			(* Spindel mit Ausfahrgeschwindigkeit *)
			IF ptrTAxisS^.T_CtrleSingle.xNotMoving THEN
				ptrTAxisS^.T_CtrleSingle.iFunction:=6;	(* Move Velocity *)
			ELSE
				ptrTAxisS^.T_CtrleSingle.iFunction:=12;	(* Move Velocity *)
			END_IF;
			ptrTAxisS^.T_CtrleSingle.lrVelocity:=T_Station_Parameter.T_StProcess.rOutfeedSpindleSpeed;
			ptrTAxisS^.T_CtrleSingle.xExecute:=TRUE;
			IF NOT(ptrTAxisBubbler^.T_CtrleDCAxis.xNotMoving) THEN
				(* Abstreifer ZU *)
				QxCylStripperClose_St1:=TRUE;
				QxCylStripperOpen_St1:=FALSE;
			END_IF
		END_IF;
		IF ptrTAxisZ^.T_LiveValue.lrActualPosition <= grZ_LoadPos THEN
			rStFct_CtrlInputWorkingSpeed:=0.0;
			T_Z_St1_Ctrle.diVelocityCommandValue:=0; (* Make sure Z axis is not moving anymore *)

			 IF ptrTAxisS^.T_CtrleSingle.xExecute AND ptrTAxisS^.T_CtrleSingle.xDone THEN
				xStFct_StartMainPrc:=FALSE;
				xStFct_InitStep:=FALSE;
				iStFct_StepPrc:=iStFct_StepPrc + 1;
			END_IF;
		END_IF;

	61: 	(* Prozess end, reset Z axis *)
		IF NOT(xStFct_InitStep) THEN
			xStFct_InitStep:=TRUE;
			xStFct_OutfeedStrokeRunning:=FALSE;
			ptrTAxisZ^.T_CtrleSingle.iFunction:=1;
			ptrTAxisZ^.T_CtrleSingle.xExecute:=TRUE;
			IF NOT(ptrTAxisBubbler^.T_CtrleDCAxis.xNotMoving) THEN
				(* Abstreifer ZU *)
				QxCylStripperClose_St1:=TRUE;
				QxCylStripperOpen_St1:=FALSE;
			END_IF
		END_IF;
		IF NOT(ptrTAxisZ^.T_CtrleSingle.xExecute) AND ptrTAxisZ^.T_CtrleSingle.xDone THEN
			xStFct_StartMainPrc:=FALSE;
			xStFct_InitStep:=FALSE;
			iStFct_StepPrc:=0;
			xStFct_SetEnd:=TRUE;
			IF xProcessDone THEN
				IF (NOT(ptrTAxisS^.T_CtrleSingle.xNotMoving) OR NOT(ptrTAxisS^.T_CtrleSingle.xDone)) AND
				     NOT((ptrTAxisS^.T_CtrleSingle.iFunction = 5) AND NOT(ptrTAxisS^.T_CtrleSingle.xDone)) AND NOT(ptrTAxisS^.T_CtrleSingle.xErr) THEN
					ptrTAxisS^.T_CtrleSingle.iFunction:=5;
					ptrTAxisS^.T_CtrleSingle.xExecute:=TRUE;
				END_IF;
			END_IF;
			(* Abstreifer AUF *)
			QxCylStripperClose_St1:=FALSE;
			QxCylStripperOpen_St1:=TRUE;
		END_IF;

		(* Dies gilt für den neuen Ablauf und setzt die Z Achse zurück auf die LadePos und gibt einen Fehler aus *)
	90:	IF (T_Station_Parameter.T_StProcess.rZ1AxisPosSwitchOAxisOff >= garPositionEndProcCalc[1])
		OR ((ptrTAxisZ^.T_LiveValue.lrActualPosition <= T_Station_Parameter.T_StProcess.rZ1AxisPosSwitchOAxisOff)
		OR (ABS(ptrTAxisZ^.T_LiveValue.lrActualPosition - T_Station_Parameter.T_StProcess.rPositionLoad) <= 10.0)) THEN
			QxFastStrokeOn_St1:=FALSE;
		END_IF;
		IF NOT(xStFct_InitStep) THEN
			xStFct_InitStep:=TRUE;
			ptrTAxisZ^.T_CtrleSingle.iFunction:=7;	(* Absolut Bewegung *)
			ptrTAxisZ^.T_CtrleSingle.lrPosition:=grZ_LoadPos;	(* AxisSlide auf BearbStartPosition setzen *)
			ptrTAxisZ^.T_CtrleSingle.lrVelocity:=rOutfeedStrokeAxisSpeed;
			ptrTAxisZ^.T_CtrleSingle.xExecute:=TRUE;
			(* Spindel mit Ausfahrgeschwindigkeit *)
			IF ptrTAxisS^.T_CtrleSingle.xNotMoving THEN
				ptrTAxisS^.T_CtrleSingle.iFunction:=6;	(* Move Velocity *)
			ELSE
				ptrTAxisS^.T_CtrleSingle.iFunction:=12;	(* Move Velocity *)
			END_IF;
			ptrTAxisS^.T_CtrleSingle.lrVelocity:=T_Station_Parameter.T_StProcess.rOutfeedSpindleSpeed;
			ptrTAxisS^.T_CtrleSingle.xExecute:=TRUE;
			IF NOT(ptrTAxisBubbler^.T_CtrleDCAxis.xNotMoving) THEN
				(* Abstreifer ZU *)
				QxCylStripperClose_St1:=TRUE;
				QxCylStripperOpen_St1:=FALSE;
			END_IF
		END_IF;
		IF NOT(ptrTAxisZ^.T_CtrleSingle.xExecute) AND ptrTAxisZ^.T_CtrleSingle.xDone AND
		     NOT(ptrTAxisS^.T_CtrleSingle.xExecute) AND ptrTAxisS^.T_CtrleSingle.xDone THEN
			xStFct_StartMainPrc:=FALSE;
			xStFct_InitStep:=FALSE;
			iStFct_StepPrc:=iStFct_StepPrc + 1;
		END_IF;

	91:	(* Abstreifer AUF *)
		QxCylStripperClose_St1:=FALSE;
		QxCylStripperOpen_St1:=TRUE;
		QxFastStrokeOn_St1:=FALSE;
		xStFct_HardwareError:=TRUE;
		diStFct_TmpErrorNr:=44;		(* Beim zylindrischer Teil wurde die Max EndPos erreicht *)

	END_CASE;
END_IF;
(******************************************************************************************************************************************)
(****************************			             Stationsfunktion Parallelablauf                                       *****************************)
(******************************************************************************************************************************************)

(******************************************************************************************************************************************)
(****************************				     Stationsfunktion Endprozedur                                    *****************************)
(******************************************************************************************************************************************)
StationFunction_Ctrl_End;
END_ACTION
ACTION StationFunction_Fct_06_ToolRotationOFF:
(******************************************************************************************************************************************)
(****************************				           Reset Stationsfunktion                                            *****************************)
(******************************************************************************************************************************************)
StationFunction_Ctrl_Reset;
(******************************************************************************************************************************************)
(****************************			        Stationsfunktion Fehler Controller                                    *****************************)
(******************************************************************************************************************************************)
StationFunction_Ctrl_Error;
(******************************************************************************************************************************************)
(****************************				    Stationsfunktion Haupt Controller                               *****************************)
(******************************************************************************************************************************************)
StationFunction_Ctrl_Main;
(******************************************************************************************************************************************)
(****************************			         Stationsfunktion sofort Unterbrechung                           *****************************)
(******************************************************************************************************************************************)
StationFunction_Ctrl_Stop;
(******************************************************************************************************************************************)
(****************************			             Stationsfunktion Hauptablauf                                       *****************************)
(******************************************************************************************************************************************)
IF xStFct_StartMainPrc AND NOT(xStFct_SetEnd) AND NOT(xStFct_HardwareError) AND NOT(xStFct_TmpStop) THEN
	CASE iStFct_StepPrc OF
	1:	IF NOT(xStFct_InitStep) THEN
			IF NOT(ptrTAxisS^.T_CtrleSingle.xNotMoving) AND ptrTAxisS^.T_CtrleSingle.xPower THEN
				(* Die Spindel dreht, daher muss sie gestoppt werden und dann der Strom noch ausschalten *)
				iStFct_StepPrc:=iStFct_StepPrc + 1;
			ELSIF ptrTAxisS^.T_CtrleSingle.xNotMoving AND ptrTAxisS^.T_CtrleSingle.xPower THEN
				(* Die Spindel ist schon gestoppt, der Strom muss aber noch ausgeschaltet werden *)
				iStFct_StepPrc:=3;
			ELSE
				(* Die Spindel ist schon im entsprechenden Zustand, daher kann die Funktion beendet werden *)
				iStFct_StepPrc:=4;
			END_IF;
			xStFct_StartMainPrc:=FALSE;
			xStFct_InitStep:=FALSE;
		END_IF;
	2:	IF NOT(xStFct_InitStep) THEN
			xStFct_InitStep:=TRUE;
			ptrTAxisS^.T_CtrleSingle.iFunction:=5;
			ptrTAxisS^.T_CtrleSingle.xExecute:=TRUE;
		END_IF;
		IF NOT(ptrTAxisS^.T_CtrleSingle.xExecute) AND ptrTAxisS^.T_CtrleSingle.xDone AND ptrTAxisS^.T_CtrleSingle.xNotMoving THEN
			xStFct_StartMainPrc:=FALSE;
			xStFct_InitStep:=FALSE;
			iStFct_StepPrc:=iStFct_StepPrc + 1;
		END_IF;
	3:	IF NOT(xStFct_InitStep) THEN
			xStFct_InitStep:=TRUE;
			ptrTAxisS^.T_CtrleSingle.iFunction:=4;	(* Strom ausschalten *)
			ptrTAxisS^.T_CtrleSingle.xExecute:=TRUE;
		END_IF;
		IF NOT(ptrTAxisS^.T_CtrleSingle.xExecute) AND ptrTAxisS^.T_CtrleSingle.xDone AND NOT(ptrTAxisS^.T_CtrleSingle.xPower) THEN
			xStFct_StartMainPrc:=FALSE;
			xStFct_InitStep:=FALSE;
			iStFct_StepPrc:=iStFct_StepPrc + 1;
		END_IF;
	4:	xStFct_StartMainPrc:=FALSE;
		xStFct_InitStep:=FALSE;
		iStFct_StepPrc:=0;
		xStFct_SetEnd:=TRUE;
	END_CASE;
END_IF;
(******************************************************************************************************************************************)
(****************************			             Stationsfunktion Parallelablauf                                       *****************************)
(******************************************************************************************************************************************)
IF xStFct_StartPrc_Parallel AND NOT(xStFct_SetEnd) AND NOT(xStFct_HardwareError) THEN
	CASE iStFct_StepPrc_Parallel OF
	1:	iStFct_StepPrc_Parallel:=1;
		xStFct_InitStep_Parallel:=FALSE;
		xStFct_StartPrc_Parallel:=FALSE;
	END_CASE;
END_IF;
(******************************************************************************************************************************************)
(****************************				     Stationsfunktion Endprozedur                                    *****************************)
(******************************************************************************************************************************************)
StationFunction_Ctrl_End;
END_ACTION
ACTION StationFunction_Fct_07_Calibration:
(******************************************************************************************************************************************)
(****************************				           Reset Stationsfunktion                                            *****************************)
(******************************************************************************************************************************************)
StationFunction_Ctrl_Reset;
(******************************************************************************************************************************************)
(****************************			        Stationsfunktion Fehler Controller                                    *****************************)
(******************************************************************************************************************************************)
StationFunction_Ctrl_Error;
(******************************************************************************************************************************************)
(****************************				    Stationsfunktion Haupt Controller                               *****************************)
(******************************************************************************************************************************************)
StationFunction_Ctrl_Main;
(******************************************************************************************************************************************)
(****************************			         Stationsfunktion sofort Unterbrechung                           *****************************)
(******************************************************************************************************************************************)
StationFunction_Ctrl_Stop;
(******************************************************************************************************************************************)
(****************************			             Stationsfunktion Hauptablauf                                       *****************************)
(******************************************************************************************************************************************)
IF xStFct_TmpStop AND NOT(xStFct_HardwareError) THEN
	T_Station_Parameter.T_Fct_SpindleCalibration.arOffsetToolDeflection[1]:=rStFct_TmpOffsetDeflection;
	T_Station_Parameter.T_Fct_SpindleCalibration.arOffsetToolTorque[1]:=rStFct_TmpOffsetTorque;
END_IF;
IF xStFct_StartMainPrc AND NOT(xStFct_SetEnd) AND NOT(xStFct_HardwareError) AND NOT(xStFct_TmpStop) THEN
	IF ((iStFct_StepPrc >= 4) AND (iStFct_StepPrc <= 6)) OR xStFct_StartPrc_Parallel THEN
		IF ((iStFct_StepPrc >= 4) AND (iStFct_StepPrc <= 6)) THEN
			T_Station_Work.THWWorkStation.TCtrlWork.rOffsetToolDeflection:=rStFct_ForceDeflection;
		END_IF;
		IF xStFct_StartPrc_Parallel THEN
			T_Station_Work.THWWorkStation.TCtrlWork.rOffsetToolTorque:=rStFct_ForceTorque;
		END_IF;
		CASE T_ExchgParam.bToolSpindleActive OF
		1:	(* Maxon Spindel *)
			IF NOT(xStFct_DeflCalibError) AND ((rStFct_ForceDeflection < 0) OR (rStFct_ForceDeflection > (T_Station_Parameter.T_SpindleSystem.rMaxDeflectionForce + rStFct_TmpOffsetDeflection))) THEN
				xStFct_DeflCalibError:=TRUE;
				xStFct_StartMainPrc:=FALSE;
				xStFct_InitStep:=FALSE;
				iStFct_StepPrc:=7;
				T_Station_Parameter.T_Fct_SpindleCalibration.arOffsetToolDeflection[1]:=rStFct_TmpOffsetDeflection;
			END_IF;
			IF NOT(xStFct_TorqueCalibError) AND ((rStFct_ForceTorque < 0) OR (rStFct_ForceTorque > (T_Station_Parameter.T_TorqueSystem.rMaxTorque_HC + rStFct_TmpOffsetTorque))) THEN
				xStFct_TorqueCalibError:=TRUE;
				xStFct_StartMainPrc:=FALSE;
				xStFct_InitStep:=FALSE;
				iStFct_StepPrc:=7;
				T_Station_Parameter.T_Fct_SpindleCalibration.arOffsetToolTorque[1]:=rStFct_TmpOffsetTorque;
				xStFct_StartPrc_Parallel:=FALSE;
			END_IF;
		2:	(* Beckhoff Spindel L *)
			IF NOT(xStFct_DeflCalibError) AND ((rStFct_ForceDeflection < 0) OR (rStFct_ForceDeflection > (T_Station_Parameter.T_SpindleSystem_L.rMaxDeflectionForce + rStFct_TmpOffsetDeflection))) THEN
				xStFct_DeflCalibError:=TRUE;
				xStFct_StartMainPrc:=FALSE;
				xStFct_InitStep:=FALSE;
				iStFct_StepPrc:=7;
				T_Station_Parameter.T_Fct_SpindleCalibration.arOffsetToolDeflection[1]:=rStFct_TmpOffsetDeflection;
			END_IF;
		3:	(* Beckhoff Spindel M *)
			IF NOT(xStFct_DeflCalibError) AND ((rStFct_ForceDeflection < 0) OR (rStFct_ForceDeflection > (T_Station_Parameter.T_SpindleSystem_M.rMaxDeflectionForce + rStFct_TmpOffsetDeflection))) THEN
				xStFct_DeflCalibError:=TRUE;
				xStFct_StartMainPrc:=FALSE;
				xStFct_InitStep:=FALSE;
				iStFct_StepPrc:=7;
				T_Station_Parameter.T_Fct_SpindleCalibration.arOffsetToolDeflection[1]:=rStFct_TmpOffsetDeflection;
			END_IF;
		END_CASE;
	END_IF;
	IF T_Station_Work.THWWorkStation.TCtrlWork.xWorkStopToolRotation THEN
		xStFct_TmpSaveOffset:=FALSE;
		xStFct_StartMainPrc:=FALSE;
		xStFct_InitStep:=FALSE;
		iStFct_StepPrc:=0;
		xStFct_SetEnd:=TRUE;
	END_IF;
	(* Deflection Sensor ON/OFF-->Muss für 0.1s gesetzt bleiben, damit Sensor ON/OFF ist, damit Prellungen ausgeschaltet werden können *)
	IF ptrTCylToolDeflection^.T_CtrleCyl.xStatePosOn THEN
		TONStFct_DeflectionSensorOFF(IN:=FALSE);
		TONStFct_DeflectionSensorON(IN:=TRUE,PT:=T#0.05s);
		IF TONStFct_DeflectionSensorON.Q THEN
			xStFct_DeflectionSensorON:=TRUE;
		END_IF;
	ELSE
		TONStFct_DeflectionSensorON(IN:=FALSE);
		TONStFct_DeflectionSensorOFF(IN:=TRUE,PT:=T#0.05s);
		IF TONStFct_DeflectionSensorOFF.Q THEN
			xStFct_DeflectionSensorON:=FALSE;
		END_IF;
	END_IF;
	(* Toruque Sensor ON/OFF-->Muss für 0.1s gesetzt bleiben, damit Sensor ON/OFF ist, damit Prellungen ausgeschaltet werden können *)
	IF ptrTCylToolTorqueHC^.T_CtrleCyl.xStatePosOn THEN
		TONStFct_TorqueSensorOFF(IN:=FALSE);
		TONStFct_TorqueSensorON(IN:=TRUE,PT:=T#0.04s);
		IF TONStFct_TorqueSensorON.Q THEN
			xStFct_TorqueSensorON:=TRUE;
		END_IF;
	ELSE
		TONStFct_TorqueSensorON(IN:=FALSE);
		TONStFct_TorqueSensorOFF(IN:=TRUE,PT:=T#0.04s);
		IF TONStFct_TorqueSensorOFF.Q THEN
			xStFct_TorqueSensorON:=FALSE;
		END_IF;
	END_IF;
	CASE iStFct_StepPrc OF
	1:	(* Offsets während Kalibrierung auf 0 setzen, aktuelle Werte für den Fehlerfall temporär ziwschen speichern*)
		xStFct_TmpSaveOffset:=TRUE;
		TONStFct_DeflectionSensorON(IN:=FALSE);
		TONStFct_DeflectionSensorOFF(IN:=FALSE);
		TONStFct_TorqueSensorON(IN:=FALSE);
		TONStFct_TorqueSensorOFF(IN:=FALSE);
		xStFct_DeflectionSensorON:=FALSE;
		xStFct_TorqueSensorON:=FALSE;
		IF  (T_Station_Parameter.T_Fct_SpindleCalibration.arOffsetToolDeflection[1] < 0) THEN
			T_Station_Parameter.T_Fct_SpindleCalibration.arOffsetToolDeflection[1]:=2.0;
			rStFct_TmpOffsetDeflection:= 2.0;
		ELSE
			rStFct_TmpOffsetDeflection:= T_Station_Parameter.T_Fct_SpindleCalibration.arOffsetToolDeflection[1];
		END_IF;
		IF (T_Station_Parameter.T_Fct_SpindleCalibration.arOffsetToolTorque[1] < 0) THEN
			T_Station_Parameter.T_Fct_SpindleCalibration.arOffsetToolTorque[1]:=2.0;
			rStFct_TmpOffsetTorque:= 2.0;
		ELSE
			rStFct_TmpOffsetTorque:= T_Station_Parameter.T_Fct_SpindleCalibration.arOffsetToolTorque[1];
		END_IF;
		xStFct_DeflCalibError:=FALSE;
		xStFct_TorqueCalibError:=FALSE;
		IF NOT(xStFct_InitStep) THEN
			(* Falls die Spindel nicht bestromt ist, dann wird der Motorstrom eingeschaltet *)
			IF NOT(ptrTAxisS^.T_CtrleSingle.xPower) THEN
				ptrTAxisS^.T_CtrleSingle.iFunction:=3;	(* Strom einschalten *)
				ptrTAxisS^.T_CtrleSingle.xExecute:=TRUE;
			END_IF;
			(* Zylinder für Überlast Drehmoment *)
			ptrTCylToolTorqueOverload^.T_CtrleCyl.iFunction:=2;
			ptrTCylToolTorqueOverload^.T_Config.tDelayOn:=T#0.2s;
			CASE T_ExchgParam.bToolSpindleActive OF
			1:	(* Maxon Spindel *)
				ptrTCylToolTorqueOverload^.T_CtrleCyl.T_Analog.rForceIn:=T_Station_Parameter.T_TorqueSystem.rMaxTorque_HCOver;	(* Dieser Zylinder muss aktiviert sein, anderenfalls führt es zu Probleme mit der Kalibrierung wegem auskoppeln der Spindel *)
			END_CASE;
			ptrTCylToolTorqueOverload^.T_CtrleCyl.xExecute:=(T_ExchgParam.bToolSpindleActive = 1);		(* nur ausführen wenn Maxon Spindel aktiv ist *)
			xStFct_InitStep:=TRUE;
		END_IF;
		IF NOT(ptrTAxisS^.T_CtrleSingle.xExecute) AND ptrTAxisS^.T_CtrleSingle.xDone AND ptrTAxisS^.T_CtrleSingle.xPower AND
		     NOT(ptrTCylToolTorqueOverload^.T_CtrleCyl.xExecute) AND ptrTCylToolTorqueOverload^.T_CtrleCyl.xDone THEN
			IF T_Station_Work.THWWorkStation.TCtrlWork.xActiveCalibrateToolDeflection THEN
				FOR iStFct_ii:=5 TO 2 BY -1 DO
					T_Station_Parameter.T_Fct_SpindleCalibration.arOffsetToolDeflection[iStFct_ii]:=T_Station_Parameter.T_Fct_SpindleCalibration.arOffsetToolDeflection[iStFct_ii-1];
				END_FOR;
			END_IF;
			IF T_Station_Work.THWWorkStation.TCtrlWork.xActiveCalibrateToolTorque THEN
				FOR iStFct_ii:=5 TO 2 BY -1 DO
					T_Station_Parameter.T_Fct_SpindleCalibration.arOffsetToolTorque[iStFct_ii]:=T_Station_Parameter.T_Fct_SpindleCalibration.arOffsetToolTorque[iStFct_ii-1];
				END_FOR;
			END_IF;
			xStFct_StartMainPrc:=FALSE;
			xStFct_InitStep:=FALSE;
			iStFct_StepPrc:=iStFct_StepPrc + 1;
		END_IF;
	2:	IF NOT(xStFct_InitStep) THEN
			xStFct_InitStep:=TRUE;
			IF ptrTAxisS^.T_CtrleSingle.xNotMoving THEN
				ptrTAxisS^.T_CtrleSingle.iFunction:=6;	(* Move Velocity *)
			ELSE
				ptrTAxisS^.T_CtrleSingle.iFunction:=12;	(* Move Velocity with new velocity *)
			END_IF;
			ptrTAxisS^.T_CtrleSingle.lrVelocity:=T_Station_Parameter.T_OnlineChange.rWorkingSpindleSpeed;
			ptrTAxisS^.T_CtrleSingle.xExecute:=TRUE;
		END_IF;
		IF NOT(ptrTAxisS^.T_CtrleSingle.xExecute) AND ptrTAxisS^.T_CtrleSingle.xDone AND NOT(ptrTAxisS^.T_CtrleSingle.xNotMoving) THEN
			rStFct_ForceDeflection:=rStFct_TmpOffsetDeflection;
			rStFct_ForceTorque:=rStFct_TmpOffsetTorque;
			IF T_Station_Work.THWWorkStation.TCtrlWork.xActiveCalibrateToolDeflection THEN
				T_Station_Parameter.T_Fct_SpindleCalibration.arOffsetToolDeflection[1]:=0.0;
			END_IF;
			IF T_Station_Work.THWWorkStation.TCtrlWork.xActiveCalibrateToolTorque THEN
				T_Station_Parameter.T_Fct_SpindleCalibration.arOffsetToolTorque[1]:=0.0;
			END_IF;
			xStFct_StartMainPrc:=FALSE;
			xStFct_InitStep:=FALSE;
			iStFct_StepPrc:=iStFct_StepPrc + 1;
		END_IF;
	(* Überprüfe zuerst ob die Sensorik in Ordnung ist *)
	3:	IF NOT(xStFct_InitStep) THEN
			xStFct_InitStep:=TRUE;
			IF T_Station_Work.THWWorkStation.TCtrlWork.xActiveCalibrateToolDeflection THEN
				(* Zylinder für Auslenkung-->ausschalten *)
				ptrTCylToolDeflection^.T_CtrleCyl.iFunction:=1;
				ptrTCylToolDeflection^.T_CtrleCyl.T_Analog.tDelayActiv:=T#0s;
				ptrTCylToolDeflection^.T_Config.tDelayOff:=T#0.3s;
				ptrTCylToolDeflection^.T_Config.xCtrlePosOff:=FALSE;
				ptrTCylToolDeflection^.T_CtrleCyl.T_Analog.rForceIn:=0.0;
				ptrTCylToolDeflection^.T_CtrleCyl.xExecute:=TRUE;
			END_IF;
			IF T_Station_Work.THWWorkStation.TCtrlWork.xActiveCalibrateToolTorque THEN
				(* Zylinder für Drehmoment-->ausschalten *)
				ptrTCylToolTorqueHC^.T_CtrleCyl.iFunction:=1;
				ptrTCylToolTorqueHC^.T_CtrleCyl.T_Analog.tDelayActiv:=T#0s;
				ptrTCylToolTorqueHC^.T_Config.tDelayOff:=T#1.0s;
				ptrTCylToolTorqueHC^.T_Config.xCtrlePosOff:=FALSE;
				ptrTCylToolTorqueHC^.T_CtrleCyl.T_Analog.rForceIn:=0.0;
				ptrTCylToolTorqueHC^.T_CtrleCyl.xExecute:=TRUE;
			END_IF;
			xStFct_ToolTorqueCheckedOK:=FALSE;
		END_IF;
		IF ptrTCylToolTorqueHC^.T_CtrleCyl.xStatePosOn THEN
			xStFct_ToolTorqueCheckedOK:=TRUE;
			ptrTCylToolTorqueHC^.T_CtrleCyl.xReset:=TRUE;
		END_IF;
		IF NOT(ptrTCylToolDeflection^.T_CtrleCyl.xExecute) AND ptrTCylToolDeflection^.T_CtrleCyl.xDone AND
		     NOT(ptrTCylToolTorqueHC^.T_CtrleCyl.xExecute) AND ptrTCylToolTorqueHC^.T_CtrleCyl.xDone THEN
			xStFct_CheckState1:=ptrTCylToolDeflection^.T_CtrleCyl.xStatePosOn;
			xStFct_CheckState2:=ptrTCylToolTorqueHC^.T_CtrleCyl.xStatePosOn OR xStFct_ToolTorqueCheckedOK;
			xStFct_CheckActive1:=T_Station_Work.THWWorkStation.TCtrlWork.xActiveCalibrateToolDeflection;
			xStFct_CheckActive2:=T_Station_Work.THWWorkStation.TCtrlWork.xActiveCalibrateToolTorque;
			IF (xStFct_CheckState1 AND xStFct_CheckState2) OR
			     (NOT(xStFct_CheckState1) AND NOT(xStFct_CheckActive1) AND xStFct_CheckState2 AND xStFct_CheckActive2) OR
			     (xStFct_CheckState1 AND xStFct_CheckActive1 AND NOT(xStFct_CheckState2) AND NOT(xStFct_CheckActive2)) THEN
				IF xStFct_CheckActive1 THEN
					iStFct_StepPrc:=iStFct_StepPrc + 1;
					xStFct_FirstTime:=TRUE;
				ELSE
					iStFct_StepPrc:=7;
				END_IF;
				IF xStFct_CheckActive2 THEN
					xStFct_StartPrc_Parallel:=TRUE;		(* Start Parallel Prozedur *)
					xStFct_FirstTimeTorque:=TRUE;
				END_IF;
				xStFct_StartMainPrc:=FALSE;
				xStFct_InitStep:=FALSE;
			ELSE
				IF xStFct_CheckActive1 AND xStFct_CheckActive2 THEN
					IF NOT(xStFct_CheckState1) AND xStFct_CheckState2 AND xStFct_CheckActive1 THEN
						diStFct_TmpErrorNr:=38;		(* Kalibrierung-->ZylWzAuslenkung Zylinder blockiert *)
					ELSIF xStFct_CheckState1 AND NOT(xStFct_CheckState2) AND xStFct_CheckActive2 THEN
						diStFct_TmpErrorNr:=39;		(* Kalibrierung-->ZylWzDrehmHC Zylinder blockiert *)
					ELSE
						diStFct_TmpErrorNr:=40;		(* Kalibrierung-->ZylWzAuslenkung+ZylWzDrehmHC Zylinder blockiert *)
					END_IF;
					T_Station_Parameter.T_Fct_SpindleCalibration.arOffsetToolDeflection[1]:=rStFct_TmpOffsetDeflection;
					T_Station_Parameter.T_Fct_SpindleCalibration.arOffsetToolTorque[1]:=rStFct_TmpOffsetTorque;
					xStFct_HardwareError:=TRUE;
					RETURN;
				ELSE
					IF NOT(xStFct_CheckState1) AND xStFct_CheckActive1 THEN
						diStFct_TmpErrorNr:=38;		(* Kalibrierung-->ZylWzAuslenkung Zylinder blockiert *)
					ELSIF NOT(xStFct_CheckState2) AND xStFct_CheckActive2 THEN
						diStFct_TmpErrorNr:=39;		(* Kalibrierung-->ZylWzDrehmHC Zylinder blockiert *)
					END_IF;
					T_Station_Parameter.T_Fct_SpindleCalibration.arOffsetToolDeflection[1]:=rStFct_TmpOffsetDeflection;
					T_Station_Parameter.T_Fct_SpindleCalibration.arOffsetToolTorque[1]:=rStFct_TmpOffsetTorque;
					xStFct_HardwareError:=TRUE;
				END_IF;
			END_IF;
		END_IF;
	4:	IF NOT(xStFct_InitStep) THEN
			xStFct_InitStep:=TRUE;
			xStFct_SetForceToolDeflection:=TRUE;
		END_IF;
		IF NOT(xStFct_SetForceToolDeflection) THEN
			IF NOT(xStFct_DeflectionSensorON) THEN
				IF NOT(xStFct_FirstTime) THEN
					xStFct_StartMainPrc:=FALSE;
					xStFct_InitStep:=FALSE;
					iStFct_StepPrc:=iStFct_StepPrc + 1;
					xStFct_FirstTime:=TRUE;
				ELSE
					xStFct_FirstTime:=FALSE;
					rStFct_ForceDeflection:=rStFct_ForceDeflection + 0.05;
					xStFct_InitStep:=FALSE;
				END_IF;
			ELSE
				rStFct_ForceDeflection:=rStFct_ForceDeflection + 0.1;
				xStFct_InitStep:=FALSE;
			END_IF;
		END_IF;
	5:	IF NOT(xStFct_InitStep) THEN
			xStFct_InitStep:=TRUE;
			xStFct_SetForceToolDeflection:=TRUE;
		END_IF;
		IF NOT(xStFct_SetForceToolDeflection) THEN
			IF NOT(xStFct_DeflectionSensorON) THEN
				rStFct_ForceDeflection:=rStFct_ForceDeflection - 0.05;
				xStFct_InitStep:=FALSE;
			ELSE
				IF NOT(xStFct_FirstTime) THEN
					xStFct_StartMainPrc:=FALSE;
					xStFct_InitStep:=FALSE;
					iStFct_StepPrc:=iStFct_StepPrc + 1;
					xStFct_FirstTime:=TRUE;
				ELSE
					xStFct_FirstTime:=FALSE;
					rStFct_ForceDeflection:=rStFct_ForceDeflection - 0.03;
					xStFct_InitStep:=FALSE;
				END_IF;
			END_IF;
		END_IF;
	6:	IF NOT(xStFct_InitStep) THEN
			xStFct_InitStep:=TRUE;
			xStFct_SetForceToolDeflection:=TRUE;
		END_IF;
		IF NOT(xStFct_SetForceToolDeflection) THEN
			IF NOT(xStFct_DeflectionSensorON) THEN
				IF NOT(xStFct_FirstTime) THEN
					T_Station_Work.THWWorkStation.TCtrlWork.rOffsetToolDeflection:=rStFct_ForceDeflection;
					T_Station_Parameter.T_Fct_SpindleCalibration.arOffsetToolDeflection[1]:=rStFct_ForceDeflection;
					xStFct_SetForceToolDeflection:=TRUE;
					rStFct_ForceDeflection:=T_Station_Parameter.T_OnlineChange.rForceDeflection;
					xStFct_StartMainPrc:=FALSE;
					xStFct_InitStep:=FALSE;
					iStFct_StepPrc:=iStFct_StepPrc + 1;
				ELSE
					xStFct_FirstTime:=FALSE;
					rStFct_ForceDeflection:=rStFct_ForceDeflection + 0.01;
					xStFct_InitStep:=FALSE;
				END_IF;
			ELSE
				rStFct_ForceDeflection:=rStFct_ForceDeflection + 0.01;
				xStFct_InitStep:=FALSE;
			END_IF;
		END_IF;
	7:	IF NOT(xStFct_InitStep) THEN
			IF NOT(xStFct_StartPrc_Parallel) THEN
				xStFct_InitStep:=TRUE;
				IF T_Station_Work.THWWorkStation.TCtrlWork.xStopToolRotation THEN
					T_Station_Work.THWWorkStation.TCtrlWork.xStopToolRotation:=FALSE;
					ptrTAxisS^.T_CtrleSingle.iFunction:=5;
					ptrTAxisS^.T_CtrleSingle.xExecute:=TRUE;
				ELSE
					iStFct_StepPrc:=iStFct_StepPrc + 2;
					xStFct_StartMainPrc:=FALSE;
					xStFct_InitStep:=FALSE;
					RETURN;
				END_IF;
			END_IF;
		END_IF;
		IF NOT(ptrTAxisS^.T_CtrleSingle.xExecute) AND ptrTAxisS^.T_CtrleSingle.xDone AND ptrTAxisS^.T_CtrleSingle.xNotMoving AND NOT(xStFct_StartPrc_Parallel) THEN
			xStFct_StartMainPrc:=FALSE;
			xStFct_InitStep:=FALSE;
			iStFct_StepPrc:=iStFct_StepPrc + 1;
		END_IF;
	8:	IF NOT(xStFct_InitStep) THEN
			xStFct_InitStep:=TRUE;
			ptrTAxisS^.T_CtrleSingle.iFunction:=4;	(* Strom ausschalten *)
			ptrTAxisS^.T_CtrleSingle.xExecute:=TRUE;
		END_IF;
		IF NOT(ptrTAxisS^.T_CtrleSingle.xExecute) AND ptrTAxisS^.T_CtrleSingle.xDone AND NOT(ptrTAxisS^.T_CtrleSingle.xPower) THEN
			xStFct_StartMainPrc:=FALSE;
			xStFct_InitStep:=FALSE;
			iStFct_StepPrc:=iStFct_StepPrc + 1;
		END_IF;
	9:	IF NOT(xStFct_StartPrc_Parallel) AND NOT(xStFct_SetForceToolDeflection) THEN
			IF xStFct_DeflCalibError OR xStFct_TorqueCalibError THEN
				IF xStFct_DeflCalibError AND NOT(xStFct_TorqueCalibError) THEN
					diStFct_TmpErrorNr:=6;		(* Kalibrierung-->ZylWzAuslenkung Sensor fehlerhaft *)
				ELSIF NOT(xStFct_DeflCalibError) AND xStFct_TorqueCalibError THEN
					diStFct_TmpErrorNr:=7;		(* Kalibrierung-->ZylWzDrehmHC Sensor fehlerhaft *)
				ELSE
					diStFct_TmpErrorNr:=8;		(* Kalibrierung-->ZylWzAuslenkung+ZylWzDrehmHC Sensor fehlerhaft *)
				END_IF;
				T_Station_Parameter.T_Fct_SpindleCalibration.arOffsetToolDeflection[1]:=rStFct_TmpOffsetDeflection;
				T_Station_Parameter.T_Fct_SpindleCalibration.arOffsetToolTorque[1]:=rStFct_TmpOffsetTorque;
				xStFct_HardwareError:=TRUE;
				RETURN;
			END_IF;
			xStFct_TmpSaveOffset:=FALSE;
			xStFct_StartMainPrc:=FALSE;
			xStFct_InitStep:=FALSE;
			iStFct_StepPrc:=0;
			xStFct_SetEnd:=TRUE;
		END_IF;
	END_CASE;
END_IF;
(******************************************************************************************************************************************)
(****************************			             Stationsfunktion Parallelablauf                                       *****************************)
(******************************************************************************************************************************************)
IF xStFct_StartPrc_Parallel AND NOT(xStFct_SetEnd) AND NOT(xStFct_HardwareError) THEN
	CASE iStFct_StepPrc_Parallel OF
	1:	IF NOT(xStFct_InitStep_Parallel) THEN
			xStFct_InitStep_Parallel:=TRUE;
			xStFct_SetForceToolTorque:=TRUE;
		END_IF;
		IF NOT(xStFct_SetForceToolTorque) THEN
			IF NOT(xStFct_TorqueSensorON) THEN
				IF NOT(xStFct_FirstTimeTorque) THEN
					xStFct_FirstTimeTorque:=TRUE;
					xStFct_InitStep_Parallel:=FALSE;
					iStFct_StepPrc_Parallel:=iStFct_StepPrc_Parallel + 1;
				ELSE
					xStFct_FirstTimeTorque:=FALSE;
					rStFct_ForceTorque:=rStFct_ForceTorque + 0.05;
					xStFct_InitStep_Parallel:=FALSE;
				END_IF;
			ELSE
				rStFct_ForceTorque:=rStFct_ForceTorque + 0.1;
				xStFct_InitStep_Parallel:=FALSE;
			END_IF;
		END_IF;
	2:	IF NOT(xStFct_InitStep_Parallel) THEN
			xStFct_InitStep_Parallel:=TRUE;
			xStFct_SetForceToolTorque:=TRUE;
		END_IF;
		IF NOT(xStFct_SetForceToolTorque) THEN
			IF NOT(xStFct_TorqueSensorON) THEN
				rStFct_ForceTorque:=rStFct_ForceTorque - 0.05;
				xStFct_InitStep_Parallel:=FALSE;
			ELSE
				IF NOT(xStFct_FirstTimeTorque) THEN
					xStFct_FirstTimeTorque:=TRUE;
					xStFct_InitStep_Parallel:=FALSE;
					iStFct_StepPrc_Parallel:=iStFct_StepPrc_Parallel + 1;
				ELSE
					xStFct_FirstTimeTorque:=FALSE;
					rStFct_ForceTorque:=rStFct_ForceTorque - 0.03;
					xStFct_InitStep_Parallel:=FALSE;
				END_IF;
			END_IF;
		END_IF;
	3:	IF NOT(xStFct_InitStep_Parallel) THEN
			xStFct_InitStep_Parallel:=TRUE;
			xStFct_SetForceToolTorque:=TRUE;
		END_IF;
		IF NOT(xStFct_SetForceToolTorque) THEN
			IF NOT(xStFct_TorqueSensorON) THEN
				IF NOT(xStFct_FirstTimeTorque) THEN
					T_Station_Work.THWWorkStation.TCtrlWork.rOffsetToolTorque:=rStFct_ForceTorque;
					T_Station_Parameter.T_Fct_SpindleCalibration.arOffsetToolTorque[1]:=rStFct_ForceTorque;
					xStFct_SetForceToolTorque:=TRUE;
					rStFct_ForceTorque:=T_Station_Parameter.T_OnlineChange.rTorqueLevelHC;
					iStFct_StepPrc_Parallel:=1;
					xStFct_InitStep_Parallel:=FALSE;
					xStFct_StartPrc_Parallel:=FALSE;
				ELSE
					xStFct_FirstTimeTorque:=FALSE;
					rStFct_ForceTorque:=rStFct_ForceTorque + 0.01;
					xStFct_InitStep_Parallel:=FALSE;
				END_IF;
			ELSE
				rStFct_ForceTorque:=rStFct_ForceTorque + 0.01;
				xStFct_InitStep_Parallel:=FALSE;
			END_IF;
		END_IF;
	END_CASE;
END_IF;
IF xStFct_SetForceToolDeflection THEN
	CASE iStFct_StepSetForceToolDeflection OF
		1:	ptrTCylToolDeflection^.T_CtrleCyl.iFunction:=2;
			ptrTCylToolDeflection^.T_CtrleCyl.T_Analog.tDelayActiv:=T#0s;
			ptrTCylToolDeflection^.T_Config.tDelayOn:=T#0.15s;
			ptrTCylToolDeflection^.T_Config.xCtrlePosOn:=FALSE;
			ptrTCylToolDeflection^.T_CtrleCyl.T_Analog.rForceIn:=rStFct_ForceDeflection;
			ptrTCylToolDeflection^.T_CtrleCyl.xExecute:=TRUE;
			iStFct_StepSetForceToolDeflection:=iStFct_StepSetForceToolDeflection + 1;
		2:	IF NOT(ptrTCylToolDeflection^.T_CtrleCyl.xExecute) AND ptrTCylToolDeflection^.T_CtrleCyl.xDone THEN
				xStFct_SetForceToolDeflection:=FALSE;
				iStFct_StepSetForceToolDeflection:=1;
			END_IF;
	END_CASE;
ELSE
	iStFct_StepSetForceToolDeflection:=1;
END_IF;
IF xStFct_SetForceToolTorque THEN
	CASE iStFct_StepSetForceToolTorque OF
		1:	ptrTCylToolTorqueHC^.T_CtrleCyl.iFunction:=2;
			ptrTCylToolTorqueHC^.T_CtrleCyl.T_Analog.tDelayActiv:=T#0s;
			ptrTCylToolTorqueHC^.T_Config.tDelayOn:=T#0.15s;
			ptrTCylToolTorqueHC^.T_Config.xCtrlePosOn:=FALSE;
			ptrTCylToolTorqueHC^.T_CtrleCyl.T_Analog.rForceIn:=rStFct_ForceTorque;
			ptrTCylToolTorqueHC^.T_CtrleCyl.xExecute:=TRUE;
			iStFct_StepSetForceToolTorque:=iStFct_StepSetForceToolTorque + 1;
		2:	IF NOT(ptrTCylToolTorqueHC^.T_CtrleCyl.xExecute) AND ptrTCylToolTorqueHC^.T_CtrleCyl.xDone THEN
				xStFct_SetForceToolTorque:=FALSE;
				iStFct_StepSetForceToolTorque:=1;
			END_IF;
	END_CASE;
ELSE
	iStFct_StepSetForceToolTorque:=1;
END_IF;
(******************************************************************************************************************************************)
(****************************				     Stationsfunktion Endprozedur                                    *****************************)
(******************************************************************************************************************************************)
StationFunction_Ctrl_End;
END_ACTION
ACTION StationFunction_Fct_07_Calibration2:
(******************************************************************************************************************************************)
(****************************				           Reset Stationsfunktion                                            *****************************)
(******************************************************************************************************************************************)
StationFunction_Ctrl_Reset;
(******************************************************************************************************************************************)
(****************************			        Stationsfunktion Fehler Controller                                    *****************************)
(******************************************************************************************************************************************)
StationFunction_Ctrl_Error;
(******************************************************************************************************************************************)
(****************************				    Stationsfunktion Haupt Controller                               *****************************)
(******************************************************************************************************************************************)
StationFunction_Ctrl_Main;
(******************************************************************************************************************************************)
(****************************			         Stationsfunktion sofort Unterbrechung                           *****************************)
(******************************************************************************************************************************************)
StationFunction_Ctrl_Stop;
(******************************************************************************************************************************************)
(****************************			             Stationsfunktion Hauptablauf                                       *****************************)
(******************************************************************************************************************************************)
IF xStFct_TmpStop AND NOT(xStFct_HardwareError) THEN
	T_Station_Parameter.T_Fct_SpindleCalibration.arOffsetToolDeflection[1]:=rStFct_TmpOffsetDeflection;
	T_Station_Parameter.T_Fct_SpindleCalibration.arOffsetToolTorque[1]:=rStFct_TmpOffsetTorque;
END_IF;
IF xStFct_StartMainPrc AND NOT(xStFct_SetEnd) AND NOT(xStFct_HardwareError) AND NOT(xStFct_TmpStop) THEN
	IF ((iStFct_StepPrc >= 4) AND (iStFct_StepPrc <= 6)) OR xStFct_StartPrc_Parallel THEN
		IF ((iStFct_StepPrc >= 4) AND (iStFct_StepPrc <= 6)) THEN
			T_Station_Work.THWWorkStation.TCtrlWork.rOffsetToolDeflection:=rStFct_ForceDeflection;
		END_IF;
		IF xStFct_StartPrc_Parallel THEN
			T_Station_Work.THWWorkStation.TCtrlWork.rOffsetToolTorque:=rStFct_ForceTorque;
		END_IF;
		IF NOT(xStFct_DeflCalibError) AND ((rStFct_ForceDeflection < 0) OR (rStFct_ForceDeflection > (T_Station_Parameter.T_SpindleSystem.rMaxDeflectionForce + rStFct_TmpOffsetDeflection))) THEN
			xStFct_DeflCalibError:=TRUE;
			xStFct_StartMainPrc:=FALSE;
			xStFct_InitStep:=FALSE;
			iStFct_StepPrc:=7;
			T_Station_Parameter.T_Fct_SpindleCalibration.arOffsetToolDeflection[1]:=rStFct_TmpOffsetDeflection;
		END_IF;
	END_IF;
	IF T_Station_Work.THWWorkStation.TCtrlWork.xWorkStopToolRotation THEN
		T_Station_Parameter.T_Fct_SpindleCalibration.arOffsetToolDeflection[1]:=rStFct_TmpOffsetDeflection;
		T_Station_Parameter.T_Fct_SpindleCalibration.arOffsetToolTorque[1]:=rStFct_TmpOffsetTorque;
		xStFct_TmpSaveOffset:=FALSE;
		xStFct_StartMainPrc:=FALSE;
		xStFct_InitStep:=FALSE;
		iStFct_StepPrc:=0;
		xStFct_SetEnd:=TRUE;
	END_IF;
	(* Deflection Sensor ON/OFF-->Muss für 0.1s gesetzt bleiben, damit Sensor ON/OFF ist, damit Prellungen ausgeschaltet werden können *)
	IF ptrTCylToolDeflection^.T_CtrleCyl.xStatePosOn THEN
		TONStFct_DeflectionSensorOFF(IN:=FALSE);
		TONStFct_DeflectionSensorON(IN:=TRUE,PT:=T#0.1s);
		IF TONStFct_DeflectionSensorON.Q THEN
			xStFct_DeflectionSensorON:=TRUE;
		END_IF;
	ELSE
		TONStFct_DeflectionSensorON(IN:=FALSE);
		TONStFct_DeflectionSensorOFF(IN:=TRUE,PT:=T#0.1s);
		IF TONStFct_DeflectionSensorOFF.Q THEN
			xStFct_DeflectionSensorON:=FALSE;
		END_IF;
	END_IF;
	CASE iStFct_StepPrc OF
	1:	IF gxHardwareOFF OR gxAxisOFF THEN
			iStFct_StepPrc:=9;
			RETURN;
		END_IF;
		(* Offsets während Kalibrierung auf 0 setzen, aktuelle Werte für den Fehlerfall temporär ziwschen speichern*)
		xStFct_TmpSaveOffset:=TRUE;
		TONStFct_DeflectionSensorON(IN:=FALSE);
		TONStFct_DeflectionSensorOFF(IN:=FALSE);
		xStFct_DeflectionSensorON:=FALSE;
		IF  (T_Station_Parameter.T_Fct_SpindleCalibration.arOffsetToolDeflection[1] < 0) THEN
			T_Station_Parameter.T_Fct_SpindleCalibration.arOffsetToolDeflection[1]:=6.0;
			rStFct_TmpOffsetDeflection:= 6.0;
		ELSE
			rStFct_TmpOffsetDeflection:= T_Station_Parameter.T_Fct_SpindleCalibration.arOffsetToolDeflection[1];
		END_IF;
		IF (T_Station_Parameter.T_Fct_SpindleCalibration.arOffsetToolTorque[1] < 0) THEN
			T_Station_Parameter.T_Fct_SpindleCalibration.arOffsetToolTorque[1]:=3.0;
			rStFct_TmpOffsetTorque:= 3.0;
		ELSE
			rStFct_TmpOffsetTorque:= T_Station_Parameter.T_Fct_SpindleCalibration.arOffsetToolTorque[1];
		END_IF;
		xStFct_DeflCalibError:=FALSE;
		IF NOT(xStFct_InitStep) THEN
			(* Falls die Spindel nicht bestromt ist, dann wird der Motorstrom eingeschaltet *)
			IF NOT(ptrTAxisS^.T_CtrleSingle.xPower) THEN
				xStFct_InitStep:=TRUE;
				IF T_Station_Work.THWWorkStation.TCtrlWork.xActiveCalibrateToolTorque THEN
					ptrTAxisS^.T_CtrleSingle.iFunction:=3;	(* Strom einschalten *)
					ptrTAxisS^.T_CtrleSingle.xExecute:=TRUE;
				END_IF;
			END_IF;
		END_IF;
		IF (NOT(ptrTAxisS^.T_CtrleSingle.xExecute) AND ptrTAxisS^.T_CtrleSingle.xDone AND ptrTAxisS^.T_CtrleSingle.xPower) OR NOT(T_Station_Work.THWWorkStation.TCtrlWork.xActiveCalibrateToolTorque) THEN
			IF T_Station_Work.THWWorkStation.TCtrlWork.xActiveCalibrateToolDeflection THEN
				FOR iStFct_ii:=5 TO 2 BY -1 DO
					T_Station_Parameter.T_Fct_SpindleCalibration.arOffsetToolDeflection[iStFct_ii]:=T_Station_Parameter.T_Fct_SpindleCalibration.arOffsetToolDeflection[iStFct_ii-1];
				END_FOR;
			END_IF;
			IF T_Station_Work.THWWorkStation.TCtrlWork.xActiveCalibrateToolTorque THEN
				FOR iStFct_ii:=5 TO 2 BY -1 DO
					T_Station_Parameter.T_Fct_SpindleCalibration.arOffsetToolTorque[iStFct_ii]:=T_Station_Parameter.T_Fct_SpindleCalibration.arOffsetToolTorque[iStFct_ii-1];
				END_FOR;
			END_IF;
			xStFct_StartMainPrc:=FALSE;
			xStFct_InitStep:=FALSE;
			iStFct_StepPrc:=iStFct_StepPrc + 1;
		END_IF;
	2:	IF NOT(xStFct_InitStep) THEN
			xStFct_InitStep:=TRUE;
			IF T_Station_Work.THWWorkStation.TCtrlWork.xActiveCalibrateToolTorque THEN
				ptrTAxisS^.T_CtrleSingle.iFunction:=6;	(* Move Velocity *)
				ptrTAxisS^.T_CtrleSingle.lrVelocity:=T_Station_Parameter.T_OnlineChange.rWorkingSpindleSpeed;
				ptrTAxisS^.T_CtrleSingle.xExecute:=TRUE;
			END_IF;
		END_IF;
		IF (NOT(ptrTAxisS^.T_CtrleSingle.xExecute) AND ptrTAxisS^.T_CtrleSingle.xDone AND NOT(ptrTAxisS^.T_CtrleSingle.xNotMoving)) OR NOT(T_Station_Work.THWWorkStation.TCtrlWork.xActiveCalibrateToolTorque) THEN
			rStFct_ForceDeflection:=rStFct_TmpOffsetDeflection;
			rStFct_ForceTorque:=rStFct_TmpOffsetTorque;
			IF T_Station_Work.THWWorkStation.TCtrlWork.xActiveCalibrateToolDeflection THEN
				T_Station_Parameter.T_Fct_SpindleCalibration.arOffsetToolDeflection[1]:=0.0;
			END_IF;
			IF T_Station_Work.THWWorkStation.TCtrlWork.xActiveCalibrateToolTorque THEN
				T_Station_Parameter.T_Fct_SpindleCalibration.arOffsetToolTorque[1]:=0.0;
			END_IF;
			xStFct_StartMainPrc:=FALSE;
			xStFct_InitStep:=FALSE;
			iStFct_StepPrc:=iStFct_StepPrc + 1;
		END_IF;
	(* Überprüfe zuerst ob die Sensorik in Ordnung ist *)
	3:	IF NOT(xStFct_InitStep) THEN
			xStFct_InitStep:=TRUE;
			IF T_Station_Work.THWWorkStation.TCtrlWork.xActiveCalibrateToolDeflection THEN
				(* Zylinder für Auslenkung-->ausschalten *)
				ptrTCylToolDeflection^.T_CtrleCyl.iFunction:=1;
				ptrTCylToolDeflection^.T_CtrleCyl.T_Analog.tDelayActiv:=T#0s;
				ptrTCylToolDeflection^.T_Config.tDelayOff:=T#0.3s;
				ptrTCylToolDeflection^.T_Config.xCtrlePosOff:=FALSE;
				ptrTCylToolDeflection^.T_CtrleCyl.T_Analog.rForceIn:=0.0;
				ptrTCylToolDeflection^.T_CtrleCyl.xExecute:=TRUE;
			END_IF;
		END_IF;
		IF NOT(ptrTCylToolDeflection^.T_CtrleCyl.xExecute) AND ptrTCylToolDeflection^.T_CtrleCyl.xDone THEN
			IF NOT(T_Station_Work.THWWorkStation.TCtrlWork.xActiveCalibrateToolDeflection AND NOT(ptrTCylToolDeflection^.T_CtrleCyl.xStatePosOn)) THEN
				IF T_Station_Work.THWWorkStation.TCtrlWork.xActiveCalibrateToolDeflection THEN
					iStFct_StepPrc:=iStFct_StepPrc + 1;
					xStFct_FirstTime:=TRUE;
				ELSE
					iStFct_StepPrc:=7;
				END_IF;
				IF T_Station_Work.THWWorkStation.TCtrlWork.xActiveCalibrateToolTorque THEN
					xStFct_StartPrc_Parallel:=TRUE;		(* Start Parallel Prozedur *)
				END_IF;
				xStFct_StartMainPrc:=FALSE;
				xStFct_InitStep:=FALSE;
			ELSE
				diStFct_TmpErrorNr:=35;		(* Kalibrierung-->ZylWzAuslenkung Zylinder blockiert *)
				xStFct_HardwareError:=TRUE;
				RETURN;
			END_IF;
		END_IF;
	4:	IF NOT(xStFct_InitStep) THEN
			xStFct_InitStep:=TRUE;
			xStFct_SetForceToolDeflection:=TRUE;
		END_IF;
		IF NOT(xStFct_SetForceToolDeflection) THEN
			IF NOT(xStFct_DeflectionSensorON) THEN
				IF NOT(xStFct_FirstTime) THEN
					xStFct_StartMainPrc:=FALSE;
					xStFct_InitStep:=FALSE;
					iStFct_StepPrc:=iStFct_StepPrc + 1;
					xStFct_FirstTime:=TRUE;
				ELSE
					xStFct_FirstTime:=FALSE;
					rStFct_ForceDeflection:=rStFct_ForceDeflection + 0.05;
					xStFct_InitStep:=FALSE;
				END_IF;
			ELSE
				rStFct_ForceDeflection:=rStFct_ForceDeflection + 0.1;
				xStFct_InitStep:=FALSE;
			END_IF;
		END_IF;
	5:	IF NOT(xStFct_InitStep) THEN
			xStFct_InitStep:=TRUE;
			xStFct_SetForceToolDeflection:=TRUE;
		END_IF;
		IF NOT(xStFct_SetForceToolDeflection) THEN
			IF NOT(xStFct_DeflectionSensorON) THEN
				rStFct_ForceDeflection:=rStFct_ForceDeflection - 0.05;
				xStFct_InitStep:=FALSE;
			ELSE
				IF NOT(xStFct_FirstTime) THEN
					xStFct_StartMainPrc:=FALSE;
					xStFct_InitStep:=FALSE;
					iStFct_StepPrc:=iStFct_StepPrc + 1;
					xStFct_FirstTime:=TRUE;
				ELSE
					xStFct_FirstTime:=FALSE;
					rStFct_ForceDeflection:=rStFct_ForceDeflection - 0.03;
					xStFct_InitStep:=FALSE;
				END_IF;
			END_IF;
		END_IF;
	6:	IF NOT(xStFct_InitStep) THEN
			xStFct_InitStep:=TRUE;
			xStFct_SetForceToolDeflection:=TRUE;
		END_IF;
		IF NOT(xStFct_SetForceToolDeflection) THEN
			IF NOT(xStFct_DeflectionSensorON) THEN
				IF NOT(xStFct_FirstTime) THEN
					T_Station_Work.THWWorkStation.TCtrlWork.rOffsetToolDeflection:=rStFct_ForceDeflection;
					T_Station_Parameter.T_Fct_SpindleCalibration.arOffsetToolDeflection[1]:=rStFct_ForceDeflection;
					xStFct_SetForceToolDeflection:=TRUE;
					rStFct_ForceDeflection:=T_Station_Parameter.T_OnlineChange.rForceDeflection;
					xStFct_StartMainPrc:=FALSE;
					xStFct_InitStep:=FALSE;
					iStFct_StepPrc:=iStFct_StepPrc + 1;
				ELSE
					xStFct_FirstTime:=FALSE;
					rStFct_ForceDeflection:=rStFct_ForceDeflection + 0.01;
					xStFct_InitStep:=FALSE;
				END_IF;
			ELSE
				rStFct_ForceDeflection:=rStFct_ForceDeflection + 0.01;
				xStFct_InitStep:=FALSE;
			END_IF;
		END_IF;
	7:	IF NOT(xStFct_InitStep) THEN
			IF NOT(xStFct_StartPrc_Parallel) THEN
				xStFct_InitStep:=TRUE;
				IF T_Station_Work.THWWorkStation.TCtrlWork.xStopToolRotation THEN
					T_Station_Work.THWWorkStation.TCtrlWork.xStopToolRotation:=FALSE;
					IF T_Station_Work.THWWorkStation.TCtrlWork.xActiveCalibrateToolTorque THEN
						ptrTAxisS^.T_CtrleSingle.iFunction:=5;
						ptrTAxisS^.T_CtrleSingle.xExecute:=TRUE;
					END_IF;
				ELSE
					iStFct_StepPrc:=iStFct_StepPrc + 2;
					xStFct_StartMainPrc:=FALSE;
					xStFct_InitStep:=FALSE;
					RETURN;
				END_IF;
			END_IF;
		END_IF;
		IF NOT(ptrTAxisS^.T_CtrleSingle.xExecute) AND ptrTAxisS^.T_CtrleSingle.xDone AND ptrTAxisS^.T_CtrleSingle.xNotMoving AND NOT(xStFct_StartPrc_Parallel) THEN
			xStFct_StartMainPrc:=FALSE;
			xStFct_InitStep:=FALSE;
			iStFct_StepPrc:=iStFct_StepPrc + 1;
		END_IF;
	8:	IF NOT(xStFct_InitStep) THEN
			xStFct_InitStep:=TRUE;
			ptrTAxisS^.T_CtrleSingle.iFunction:=4;	(* Strom ausschalten *)
			ptrTAxisS^.T_CtrleSingle.xExecute:=TRUE;
		END_IF;
		IF NOT(ptrTAxisS^.T_CtrleSingle.xExecute) AND ptrTAxisS^.T_CtrleSingle.xDone AND NOT(ptrTAxisS^.T_CtrleSingle.xPower) THEN
			xStFct_StartMainPrc:=FALSE;
			xStFct_InitStep:=FALSE;
			iStFct_StepPrc:=iStFct_StepPrc + 1;
		END_IF;
	9:	IF NOT(xStFct_StartPrc_Parallel) AND NOT(xStFct_SetForceToolDeflection) THEN
			IF xStFct_DeflCalibError THEN
				IF xStFct_DeflCalibError THEN
					diStFct_TmpErrorNr:=36;		(* Kalibrierung-->ZylWzAuslenkung Sensor fehlerhaft *)
				END_IF;
				xStFct_HardwareError:=TRUE;
				RETURN;
			END_IF;
			xStFct_TmpSaveOffset:=FALSE;
			xStFct_StartMainPrc:=FALSE;
			xStFct_InitStep:=FALSE;
			iStFct_StepPrc:=0;
			xStFct_SetEnd:=TRUE;
		END_IF;
	END_CASE;
END_IF;
IF xStFct_TmpSaveOffset AND xStFct_SetEnd THEN
	(* Im Fehlerfall oder die Funktion gestoppt wird muss der alte Wert wieder übergeben werden *)
	xStFct_TmpSaveOffset:=FALSE;
	T_Station_Parameter.T_Fct_SpindleCalibration.arOffsetToolDeflection[1]:=rStFct_TmpOffsetDeflection;
	T_Station_Parameter.T_Fct_SpindleCalibration.arOffsetToolTorque[1]:=rStFct_TmpOffsetTorque;
END_IF;
(******************************************************************************************************************************************)
(****************************			             Stationsfunktion Parallelablauf                                       *****************************)
(******************************************************************************************************************************************)
IF xStFct_StartPrc_Parallel AND NOT(xStFct_SetEnd) AND NOT(xStFct_HardwareError) THEN
	CASE iStFct_StepPrc_Parallel OF
	1:	IF NOT(xStFct_InitStep_Parallel) THEN
			xStFct_InitStep_Parallel:=TRUE;
			TONStFct_WaitMeasure(IN:=FALSE);
		END_IF;
		TONStFct_WaitMeasure(IN:=TRUE,PT:=T#0.2s);
		IF TONStFct_WaitMeasure.Q THEN
			TONStFct_WaitMeasure(IN:=FALSE);
			xStFct_InitStep_Parallel:=FALSE;
			iStFct_MeasuringStep:=iStFct_MeasuringStep + 1;
			IF (iStFct_MeasuringStep <= 20) THEN
				arStFct_NullPointToolTorque[iStFct_MeasuringStep]:=ptrTSensorTorque^.T_CtrleCyl.T_Analog.rPosIn;
				rStFct_ForceTorque:=ptrTSensorTorque^.T_CtrleCyl.T_Analog.rPosIn;
			ELSE
				iStFct_StepPrc_Parallel:=iStFct_StepPrc_Parallel + 1;
			END_IF;
		END_IF;
	2:	rStFct_NullPointToolTorque:=0.0;
		FOR iStFct_ii:=1 TO 20 DO
			rStFct_NullPointToolTorque:=rStFct_NullPointToolTorque + arStFct_NullPointToolTorque[iStFct_ii];
		END_FOR;
		rStFct_ForceTorque:=rStFct_NullPointToolTorque / 20.0;
		T_Station_Work.THWWorkStation.TCtrlWork.rOffsetToolTorque:=rStFct_ForceTorque;
		T_Station_Parameter.T_Fct_SpindleCalibration.arOffsetToolTorque[1]:=rStFct_ForceTorque;
		iStFct_StepPrc_Parallel:=1;
		xStFct_InitStep_Parallel:=FALSE;
		xStFct_StartPrc_Parallel:=FALSE;
	END_CASE;
ELSE
	iStFct_MeasuringStep:=0;
END_IF;
IF xStFct_SetForceToolDeflection THEN
	CASE iStFct_StepSetForceToolDeflection OF
		1:	ptrTCylToolDeflection^.T_CtrleCyl.iFunction:=2;
			ptrTCylToolDeflection^.T_CtrleCyl.T_Analog.tDelayActiv:=T#0s;
			ptrTCylToolDeflection^.T_Config.tDelayOn:=T#0.15s;
			ptrTCylToolDeflection^.T_Config.xCtrlePosOn:=FALSE;
			ptrTCylToolDeflection^.T_CtrleCyl.T_Analog.rForceIn:=rStFct_ForceDeflection;
			ptrTCylToolDeflection^.T_CtrleCyl.xExecute:=TRUE;
			iStFct_StepSetForceToolDeflection:=iStFct_StepSetForceToolDeflection + 1;
		2:	IF NOT(ptrTCylToolDeflection^.T_CtrleCyl.xExecute) AND ptrTCylToolDeflection^.T_CtrleCyl.xDone THEN
				xStFct_SetForceToolDeflection:=FALSE;
				iStFct_StepSetForceToolDeflection:=1;
			END_IF;
	END_CASE;
ELSE
	iStFct_StepSetForceToolDeflection:=1;
END_IF;
(******************************************************************************************************************************************)
(****************************				     Stationsfunktion Endprozedur                                    *****************************)
(******************************************************************************************************************************************)
StationFunction_Ctrl_End;
END_ACTION
ACTION StationFunction_Fct_08_SpindleBurnIn:
(******************************************************************************************************************************************)
(****************************				           Reset Stationsfunktion                                            *****************************)
(******************************************************************************************************************************************)
StationFunction_Ctrl_Reset;
(******************************************************************************************************************************************)
(****************************			        Stationsfunktion Fehler Controller                                    *****************************)
(******************************************************************************************************************************************)
StationFunction_Ctrl_Error;
(******************************************************************************************************************************************)
(****************************				    Stationsfunktion Haupt Controller                               *****************************)
(******************************************************************************************************************************************)
StationFunction_Ctrl_Main;
(******************************************************************************************************************************************)
(****************************			         Stationsfunktion sofort Unterbrechung                           *****************************)
(******************************************************************************************************************************************)
StationFunction_Ctrl_Stop;
(******************************************************************************************************************************************)
(****************************			             Stationsfunktion Hauptablauf                                       *****************************)
(******************************************************************************************************************************************)
IF (T_Station_Parameter.T_Fct_SpindleBurnIn.rTimeMaxActiveFunction <> 0) THEN	(* If the Time is 0, than the function is active as long as the operator does stop *)
	tStFct_MaxTimeActiveFunction:=REAL_TO_TIME(T_Station_Parameter.T_Fct_SpindleBurnIn.rTimeMaxActiveFunction * 1000);
	IF (iStFct_StepPrc > 1) AND (iStFct_StepPrc < 10) THEN
		fbStFct_TONChkMaxTimeActive(IN:=TRUE,PT:=tStFct_MaxTimeActiveFunction);
		IF fbStFct_TONChkMaxTimeActive.Q THEN
			xStFct_StartMainPrc:=FALSE;
			xStFct_InitStep:=FALSE;
			iStFct_StepPrc:=10;
		END_IF;
	END_IF;
END_IF;
tStFct_TimeSpindleActive:=REAL_TO_TIME(T_Station_Parameter.T_Fct_SpindleBurnIn.rTimeSpindleActive * 1000.0);
IF (tStFct_TimeSpindleActive = T#0s) THEN tStFct_TimeSpindleActive:=T#5s; END_IF;
tStFct_TimeSpindleInactive:=REAL_TO_TIME(T_Station_Parameter.T_Fct_SpindleBurnIn.rTimeSpindleInactive * 1000.0);
IF (tStFct_TimeSpindleInactive = T#0s) THEN tStFct_TimeSpindleInactive:=T#5s; END_IF;
IF xStFct_StartMainPrc AND NOT(xStFct_SetEnd) AND NOT(xStFct_HardwareError) AND NOT(xStFct_TmpStop) THEN
	CASE iStFct_StepPrc OF
	1:	fbStFct_TONChkMaxTimeActive(IN:=FALSE);
		IF NOT(xStFct_InitStep) THEN
			(* Falls die Spindel nicht bestromt ist, dann wird der Motorstrom eingeschaltet *)
			IF NOT(ptrTAxisS^.T_CtrleSingle.xPower) THEN
				xStFct_InitStep:=TRUE;
				ptrTAxisS^.T_CtrleSingle.iFunction:=3;	(* Strom einschalten *)
				ptrTAxisS^.T_CtrleSingle.xExecute:=TRUE;
			END_IF;
		END_IF;
		IF NOT(ptrTAxisS^.T_CtrleSingle.xExecute) AND ptrTAxisS^.T_CtrleSingle.xDone AND ptrTAxisS^.T_CtrleSingle.xPower THEN
			xStFct_StartMainPrc:=FALSE;
			xStFct_InitStep:=FALSE;
			iStFct_StepPrc:=iStFct_StepPrc + 1;
		END_IF;
	2:	IF NOT(xStFct_InitStep) THEN
			xStFct_InitStep:=TRUE;
			(* Zylinder für Auslenkung-->mit Workauslenkkraft *)
			ptrTCylToolDeflection^.T_CtrleCyl.iFunction:=2;
			ptrTCylToolDeflection^.T_Config.tDelayOn:=T#0.3s;
			ptrTCylToolDeflection^.T_CtrleCyl.T_Analog.rForceIn:=T_Station_Parameter.T_OnlineChange.rForceDeflection;
			ptrTCylToolDeflection^.T_CtrleCyl.xExecute:=TRUE;
			(* Zylinder für Drehmoment HC-->mit Schwellwert Startposition *)
			ptrTCylToolTorqueHC^.T_CtrleCyl.iFunction:=2;
			ptrTCylToolTorqueHC^.T_Config.tDelayOn:=T#0.2s;
			ptrTCylToolTorqueHC^.T_CtrleCyl.T_Analog.rForceIn:=T_Station_Parameter.T_OnlineChange.rTorqueLevelHC;
			ptrTCylToolTorqueHC^.T_CtrleCyl.xExecute:=TRUE;
			(* Zylinder für Überlast Drehmoment *)
			ptrTCylToolTorqueOverload^.T_CtrleCyl.iFunction:=2;
			ptrTCylToolTorqueOverload^.T_Config.tDelayOn:=T#0.2s;
			ptrTCylToolTorqueOverload^.T_CtrleCyl.T_Analog.rForceIn:=T_Station_Parameter.T_StProcess.rTorqueLevel_Overload;
			ptrTCylToolTorqueOverload^.T_CtrleCyl.xExecute:=TRUE;
		END_IF;
		IF NOT(ptrTCylToolDeflection^.T_CtrleCyl.xExecute) AND ptrTCylToolDeflection^.T_CtrleCyl.xDone AND
		     NOT(ptrTCylToolTorqueHC^.T_CtrleCyl.xExecute) AND ptrTCylToolTorqueHC^.T_CtrleCyl.xDone AND
		     NOT(ptrTCylToolTorqueOverload^.T_CtrleCyl.xExecute) AND ptrTCylToolTorqueOverload^.T_CtrleCyl.xDone THEN
			xStFct_StartMainPrc:=FALSE;
			xStFct_InitStep:=FALSE;
			iStFct_StepPrc:=iStFct_StepPrc + 1;
		END_IF;
	3:	IF NOT(xStFct_InitStep) THEN
			xStFct_InitStep:=TRUE;
			IF ptrTAxisS^.T_CtrleSingle.xNotMoving THEN
				ptrTAxisS^.T_CtrleSingle.iFunction:=6;	(* Move Velocity *)
			ELSE
				ptrTAxisS^.T_CtrleSingle.iFunction:=12;	(* Move Velocity *)
			END_IF;
			ptrTAxisS^.T_CtrleSingle.lrVelocity:=T_Station_Parameter.T_Fct_SpindleBurnIn.rSpindleSpeed;
			ptrTAxisS^.T_CtrleSingle.xExecute:=TRUE;
		END_IF;
		IF NOT(ptrTAxisS^.T_CtrleSingle.xExecute) AND ptrTAxisS^.T_CtrleSingle.xDone AND NOT(ptrTAxisS^.T_CtrleSingle.xNotMoving) THEN
			xStFct_StartMainPrc:=FALSE;
			xStFct_InitStep:=FALSE;
			iStFct_StepPrc:=iStFct_StepPrc + 1;
		END_IF;
	4:	IF NOT(xStFct_InitStep) THEN
			xStFct_InitStep:=TRUE;
			fbStFct_TONWaitCycle(IN:=FALSE);
		END_IF;
		fbStFct_TONWaitCycle(IN:=TRUE,PT:=tStFct_TimeSpindleActive);
		IF fbStFct_TONWaitCycle.Q THEN
			xStFct_StartMainPrc:=FALSE;
			xStFct_InitStep:=FALSE;
			iStFct_StepPrc:=iStFct_StepPrc + 1;
		END_IF;
	5:	IF NOT(xStFct_InitStep) THEN
			xStFct_InitStep:=TRUE;
			ptrTAxisS^.T_CtrleSingle.iFunction:=5;
			ptrTAxisS^.T_CtrleSingle.xExecute:=TRUE;
		END_IF;
		IF NOT(ptrTAxisS^.T_CtrleSingle.xExecute) AND ptrTAxisS^.T_CtrleSingle.xDone AND ptrTAxisS^.T_CtrleSingle.xNotMoving THEN
			xStFct_StartMainPrc:=FALSE;
			xStFct_InitStep:=FALSE;
			iStFct_StepPrc:=iStFct_StepPrc + 1;
		END_IF;
	6:	IF NOT(xStFct_InitStep) THEN
			xStFct_InitStep:=TRUE;
			fbStFct_TONWaitCycle(IN:=FALSE);
		END_IF;
		fbStFct_TONWaitCycle(IN:=TRUE,PT:=tStFct_TimeSpindleInactive);
		IF fbStFct_TONWaitCycle.Q THEN
			xStFct_StartMainPrc:=FALSE;
			xStFct_InitStep:=FALSE;
			iStFct_StepPrc:=3;
		END_IF;
	10:	IF NOT(xStFct_InitStep) THEN
			xStFct_InitStep:=TRUE;
			ptrTAxisS^.T_CtrleSingle.iFunction:=5;
			ptrTAxisS^.T_CtrleSingle.xExecute:=TRUE;
		END_IF;
		IF NOT(ptrTAxisS^.T_CtrleSingle.xExecute) AND ptrTAxisS^.T_CtrleSingle.xDone AND ptrTAxisS^.T_CtrleSingle.xNotMoving THEN
			xStFct_StartMainPrc:=FALSE;
			xStFct_InitStep:=FALSE;
			iStFct_StepPrc:=iStFct_StepPrc + 1;
		END_IF;
	11:	IF NOT(xStFct_InitStep) THEN
			xStFct_InitStep:=TRUE;
			IF ptrTAxisS^.T_CtrleSingle.xPower THEN
				ptrTAxisS^.T_CtrleSingle.iFunction:=4;	(* Strom ausschalten *)
				ptrTAxisS^.T_CtrleSingle.xExecute:=TRUE;
			END_IF;
		END_IF;
		IF NOT(ptrTAxisS^.T_CtrleSingle.xExecute) AND ptrTAxisS^.T_CtrleSingle.xDone AND NOT(ptrTAxisS^.T_CtrleSingle.xPower) THEN
			xStFct_StartMainPrc:=FALSE;
			xStFct_InitStep:=FALSE;
			iStFct_StepPrc:=0;
			xStFct_SetEnd:=TRUE;
		END_IF;
	END_CASE;
END_IF;
(******************************************************************************************************************************************)
(****************************			             Stationsfunktion Parallelablauf                                       *****************************)
(******************************************************************************************************************************************)
IF xStFct_StartPrc_Parallel AND NOT(xStFct_SetEnd) AND NOT(xStFct_HardwareError) THEN
	CASE iStFct_StepPrc_Parallel OF
	1:	iStFct_StepPrc_Parallel:=1;
		xStFct_InitStep_Parallel:=FALSE;
		xStFct_StartPrc_Parallel:=FALSE;
	END_CASE;
END_IF;
(******************************************************************************************************************************************)
(****************************				     Stationsfunktion Endprozedur                                    *****************************)
(******************************************************************************************************************************************)
StationFunction_Ctrl_End;
END_ACTION
ACTION StationFunction_Fct_09_Initial_Z_Axis:
(******************************************************************************************************************************************)
(****************************				           Reset Stationsfunktion                                            *****************************)
(******************************************************************************************************************************************)
StationFunction_Ctrl_Reset;
(******************************************************************************************************************************************)
(****************************			        Stationsfunktion Fehler Controller                                    *****************************)
(******************************************************************************************************************************************)
StationFunction_Ctrl_Error;
(******************************************************************************************************************************************)
(****************************				    Stationsfunktion Haupt Controller                               *****************************)
(******************************************************************************************************************************************)
StationFunction_Ctrl_Main;
(******************************************************************************************************************************************)
(****************************			         Stationsfunktion sofort Unterbrechung                           *****************************)
(******************************************************************************************************************************************)
StationFunction_Ctrl_Stop;
(******************************************************************************************************************************************)
(****************************			             Stationsfunktion Hauptablauf                                       *****************************)
(******************************************************************************************************************************************)
IF xStFct_StartMainPrc AND NOT(xStFct_SetEnd) AND NOT(xStFct_HardwareError) AND NOT(xStFct_TmpStop) THEN
	CASE iStFct_StepPrc OF
	1:	wStFct_Status:=0;
		IF NOT(xStFct_InitStep) THEN
			(* Falls Z Achse sich bewegt, dann wird der Motor gestoppt *)
			IF NOT(ptrTAxisZ^.T_CtrleSingle.xExecute) AND NOT(ptrTAxisZ^.T_CtrleSingle.xNotMoving) THEN
				xStFct_InitStep:=TRUE;
				ptrTAxisZ^.T_CtrleSingle.iFunction:=5;
				ptrTAxisZ^.T_CtrleSingle.xExecute:=TRUE;
			END_IF;
		END_IF;
		IF NOT(ptrTAxisZ^.T_CtrleSingle.xExecute) AND ptrTAxisZ^.T_CtrleSingle.xDone AND ptrTAxisZ^.T_CtrleSingle.xNotMoving THEN
			xStFct_StartMainPrc:=FALSE;
			xStFct_InitStep:=FALSE;
			iStFct_StepPrc:=iStFct_StepPrc + 1;
		END_IF;
	2:	IF NOT(xStFct_InitStep) THEN
			(* Falls Z Achse nicht bestromt ist, dann wird der Motorstrom eingeschaltet *)
			IF NOT(ptrTAxisZ^.T_CtrleSingle.xPower) THEN
				xStFct_InitStep:=TRUE;
				ptrTAxisZ^.T_CtrleSingle.iFunction:=3;	(* Strom einschalten *)
				ptrTAxisZ^.T_CtrleSingle.xExecute:=TRUE;
			END_IF;
		END_IF;
		IF NOT(ptrTAxisZ^.T_CtrleSingle.xExecute) AND ptrTAxisZ^.T_CtrleSingle.xDone AND ptrTAxisZ^.T_CtrleSingle.xPower THEN
			xStFct_StartMainPrc:=FALSE;
			xStFct_InitStep:=FALSE;
			iStFct_StepPrc:=iStFct_StepPrc + 1;
		END_IF;
	3:	IF NOT(xStFct_InitStep) THEN
			xStFct_InitStep:=TRUE;
			(* Zylinder für Auslenkung-->mit Workauslenkkraft *)
			ptrTCylToolDeflection^.T_CtrleCyl.iFunction:=2;
			ptrTCylToolDeflection^.T_Config.tDelayOn:=T#0.3s;
			ptrTCylToolDeflection^.T_CtrleCyl.T_Analog.rForceIn:=T_Station_Parameter.T_OnlineChange.rForceDeflection;
			ptrTCylToolDeflection^.T_CtrleCyl.xExecute:=TRUE;
			(* Zylinder für Drehmoment HC-->mit Schwellwert Startposition *)
			ptrTCylToolTorqueHC^.T_CtrleCyl.iFunction:=2;
			ptrTCylToolTorqueHC^.T_Config.tDelayOn:=T#0.2s;
			ptrTCylToolTorqueHC^.T_CtrleCyl.T_Analog.rForceIn:=T_Station_Parameter.T_OnlineChange.rTorqueLevelHC;
			ptrTCylToolTorqueHC^.T_CtrleCyl.xExecute:=TRUE;
			(* Zylinder für Überlast Drehmoment *)
			ptrTCylToolTorqueOverload^.T_CtrleCyl.iFunction:=2;
			ptrTCylToolTorqueOverload^.T_Config.tDelayOn:=T#0.2s;
			ptrTCylToolTorqueOverload^.T_CtrleCyl.T_Analog.rForceIn:=T_Station_Parameter.T_StProcess.rTorqueLevel_Overload;
			ptrTCylToolTorqueOverload^.T_CtrleCyl.xExecute:=TRUE;
		END_IF;
		IF NOT(ptrTCylToolDeflection^.T_CtrleCyl.xExecute) AND ptrTCylToolDeflection^.T_CtrleCyl.xDone AND
		     NOT(ptrTCylToolTorqueHC^.T_CtrleCyl.xExecute) AND ptrTCylToolTorqueHC^.T_CtrleCyl.xDone AND
		     NOT(ptrTCylToolTorqueOverload^.T_CtrleCyl.xExecute) AND ptrTCylToolTorqueOverload^.T_CtrleCyl.xDone THEN
			xStFct_StartMainPrc:=FALSE;
			xStFct_InitStep:=FALSE;
			iStFct_StepPrc:=iStFct_StepPrc + 1;
		END_IF;
	(* Aufsuchen des negativen Endschalter der Z Achse *)
	4:	IF NOT(xStFct_InitStep) THEN
			xStFct_InitStep:=TRUE;
			ptrTAxisZ^.T_CtrleSingle.iFunction:=6;	(* Geschwindigkeits Bewegung *)
			ptrTAxisZ^.T_CtrleSingle.lrVelocity:=T_Station_Parameter.T_AxisState.rZDetectEndSwitchSpeed * -1.0;
			ptrTAxisZ^.T_CtrleSingle.xExecute:=TRUE;
		END_IF;
		IF NOT(ptrTAxisZ^.T_CtrleSingle.xExecute) AND ptrTAxisZ^.T_CtrleSingle.xDone THEN
			xStFct_StartMainPrc:=FALSE;
			xStFct_InitStep:=FALSE;
			iStFct_StepPrc:=iStFct_StepPrc + 1;
		END_IF;
	(* Sobald der Endschalter eintrifft muss der Treiber gestoppt werden-->Achse stoppt von selbst *)
	5:	IF ptrTAxisZ^.T_CtrleSingle.xStateHWLimitNeg THEN
			xStFct_StartMainPrc:=FALSE;
			xStFct_InitStep:=FALSE;
			iStFct_StepPrc:=iStFct_StepPrc + 1;
		END_IF;
	(* Achsen Treiber wird gestoppt *)
	6:	IF NOT(xStFct_InitStep) THEN
			xStFct_InitStep:=TRUE;
			IF NOT(ptrTAxisZ^.T_CtrleSingle.xNotMoving) AND ptrTAxisZ^.T_CtrleSingle.xDone AND NOT(ptrTAxisZ^.T_CtrleSingle.xStateHWLimitNeg) THEN
				ptrTAxisZ^.T_CtrleSingle.iFunction:=5;
				ptrTAxisZ^.T_CtrleSingle.xExecute:=TRUE;
			END_IF;
		END_IF;
		IF NOT(ptrTAxisZ^.T_CtrleSingle.xExecute) AND ptrTAxisZ^.T_CtrleSingle.xDone AND ptrTAxisZ^.T_CtrleSingle.xReady AND ptrTAxisZ^.T_CtrleSingle.xPower THEN
			xStFct_StartMainPrc:=FALSE;
			xStFct_InitStep:=FALSE;
			IF ptrTAxisZ^.T_CtrleSingle.xNotMoving THEN
				iStFct_StepPrc:=iStFct_StepPrc + 1;
			END_IF;
		END_IF;
	(* Warten bis die Achse wieder bereit steht *)
	7:	IF NOT(xStFct_InitStep) THEN
			xStFct_InitStep:=TRUE;
			TONStFct_WaitAxisReady(IN:=FALSE);
		END_IF;
		TONStFct_WaitAxisReady(IN:=TRUE,PT:=T#0.5s);
		IF TONStFct_WaitAxisReady.Q THEN
			TONStFct_WaitAxisReady(IN:=FALSE);
			xStFct_StartMainPrc:=FALSE;
			xStFct_InitStep:=FALSE;
			iStFct_StepPrc:=iStFct_StepPrc + 1;
		END_IF;
	(* Bewege die Achse weg vom Endschalter bis der Endschalter nicht mehr angibt + 1mm reserve *)
	8:	IF NOT(xStFct_InitStep) THEN
			xStFct_InitStep:=TRUE;
			ptrTAxisZ^.T_CtrleSingle.iFunction:=6;	(* Geschwindigkeits Bewegung *)
			ptrTAxisZ^.T_CtrleSingle.lrVelocity:=1.0;
			ptrTAxisZ^.T_CtrleSingle.xExecute:=TRUE;
		END_IF;
		IF NOT(ptrTAxisZ^.T_CtrleSingle.xExecute) AND ptrTAxisZ^.T_CtrleSingle.xDone THEN
			xStFct_StartMainPrc:=FALSE;
			xStFct_InitStep:=FALSE;
			iStFct_StepPrc:=iStFct_StepPrc + 1;
		END_IF;
	(* Sobald der Endschalter nicht mehr bedämpft ist und 1mm gefahren wurde dann muss die Achse gestoppt werden *)
	9:	IF NOT(ptrTAxisZ^.T_CtrleSingle.xStateHWLimitNeg) THEN
			lrStFct_SaveAxisPosition:=ptrTAxisZ^.T_LiveValue.lrActualPosition;
			xStFct_StartMainPrc:=FALSE;
			xStFct_InitStep:=FALSE;
			iStFct_StepPrc:=iStFct_StepPrc + 1;
		END_IF;
	(* Abwarten bis 0.5mm nach dem Endschalter abgefahren ist und dann die Achse stoppen *)
	10:	IF (ptrTAxisZ^.T_LiveValue.lrActualPosition >= (lrStFct_SaveAxisPosition + 0.5)) THEN
			xStFct_StartMainPrc:=FALSE;
			xStFct_InitStep:=FALSE;
			iStFct_StepPrc:=iStFct_StepPrc + 1;
		END_IF;
	(* Achse muss gestoppt werden *)
	11:	IF NOT(xStFct_InitStep) THEN
			xStFct_InitStep:=TRUE;
			IF NOT(ptrTAxisZ^.T_CtrleSingle.xNotMoving) AND ptrTAxisZ^.T_CtrleSingle.xDone THEN
				ptrTAxisZ^.T_CtrleSingle.iFunction:=5;
				ptrTAxisZ^.T_CtrleSingle.xExecute:=TRUE;
			END_IF;
		END_IF;
		IF NOT(ptrTAxisZ^.T_CtrleSingle.xExecute) AND ptrTAxisZ^.T_CtrleSingle.xDone THEN
			xStFct_StartMainPrc:=FALSE;
			xStFct_InitStep:=FALSE;
			IF ptrTAxisZ^.T_CtrleSingle.xNotMoving THEN
				iStFct_StepPrc:=iStFct_StepPrc + 1;
			END_IF;
		END_IF;
	(* Übernehmen der Position *)
	12:	T_Station_Parameter.T_AxisState.rPositionNegLimitSwitchZAxis_Old:=	T_Station_Parameter.T_AxisState.rPositionNegLimitSwitchZAxis;
		T_Station_Parameter.T_AxisState.rPositionNegLimitSwitchZAxis:=		ptrTAxisZ^.T_LiveValue.lrActualPosition;
		xStFct_StartMainPrc:=FALSE;
		xStFct_InitStep:=FALSE;
		iStFct_StepPrc:=iStFct_StepPrc + 1;
	13:	xStFct_StartMainPrc:=FALSE;
		xStFct_InitStep:=FALSE;
		iStFct_StepPrc:=0;
		xStFct_SetEnd:=TRUE;
	END_CASE;
END_IF;
(******************************************************************************************************************************************)
(****************************			             Stationsfunktion Parallelablauf                                       *****************************)
(******************************************************************************************************************************************)
IF xStFct_StartPrc_Parallel AND NOT(xStFct_SetEnd) AND NOT(xStFct_HardwareError) THEN
	CASE iStFct_StepPrc_Parallel OF
	1:	iStFct_StepPrc_Parallel:=1;
		xStFct_InitStep_Parallel:=FALSE;
		xStFct_StartPrc_Parallel:=FALSE;
	END_CASE;
END_IF;
(******************************************************************************************************************************************)
(****************************				     Stationsfunktion Endprozedur                                    *****************************)
(******************************************************************************************************************************************)
StationFunction_Ctrl_End;
END_ACTION
ACTION StationFunction_Fct_10_CheckAxisBreak:
(******************************************************************************************************************************************)
(****************************				           Reset Stationsfunktion                                            *****************************)
(******************************************************************************************************************************************)
StationFunction_Ctrl_Reset;
(******************************************************************************************************************************************)
(****************************			        Stationsfunktion Fehler Controller                                    *****************************)
(******************************************************************************************************************************************)
StationFunction_Ctrl_Error;
(******************************************************************************************************************************************)
(****************************				    Stationsfunktion Haupt Controller                               *****************************)
(******************************************************************************************************************************************)
StationFunction_Ctrl_Main;
(******************************************************************************************************************************************)
(****************************			         Stationsfunktion sofort Unterbrechung                           *****************************)
(******************************************************************************************************************************************)
StationFunction_Ctrl_Stop;
(******************************************************************************************************************************************)
(****************************			             Stationsfunktion Hauptablauf                                       *****************************)
(******************************************************************************************************************************************)
IF xStFct_StartMainPrc AND NOT(xStFct_SetEnd) AND NOT(xStFct_HardwareError) AND NOT(xStFct_TmpStop) THEN
	CASE iStFct_StepPrc OF
	1:	IF NOT(xStFct_InitStep) THEN
			T_Station_Work.THWWorkStation.TCtrlWork.xBlockCheckAxisBrake:=TRUE;	(* Überwachung muss für diese Funktion ausgeschaltet werden *)
			xStFct_ZAxisBrakeBlocked:=FALSE;
			xStFct_InitStep:=TRUE;
			(* Bremszylinder für Achse Z *)
			ptrTCylBrakeReleaseZAxis^.T_CtrleCyl.iFunction:=1;
			ptrTCylBrakeReleaseZAxis^.T_CtrleCyl.xExecute:=TRUE;
		END_IF;
		IF NOT(ptrTCylBrakeReleaseZAxis^.T_CtrleCyl.xExecute) AND ptrTCylBrakeReleaseZAxis^.T_CtrleCyl.xDone THEN
			IF ptrTCylBrakeReleaseZAxis^.T_CtrleCyl.xStatePosOn THEN
				xStFct_ZAxisBrakeBlocked:=TRUE;	(* Achsenbremse ist blockiert *)
			END_IF;
			xStFct_StartMainPrc:=FALSE;
			xStFct_InitStep:=FALSE;
			iStFct_StepPrc:=iStFct_StepPrc + 1;
		END_IF;
	2:	IF NOT(xStFct_InitStep) THEN
			xStFct_InitStep:=TRUE;
			(* Bremszylinder für Achse Z *)
			ptrTCylBrakeReleaseZAxis^.T_CtrleCyl.iFunction:=2;
			ptrTCylBrakeReleaseZAxis^.T_CtrleCyl.xExecute:=TRUE;
		END_IF;
		IF NOT(ptrTCylBrakeReleaseZAxis^.T_CtrleCyl.xExecute) AND ptrTCylBrakeReleaseZAxis^.T_CtrleCyl.xDone THEN
			IF NOT(ptrTCylBrakeReleaseZAxis^.T_CtrleCyl.xStatePosOn) THEN
				xStFct_ZAxisBrakeBlocked:=TRUE;	(* Sensor evtl nicht richtig eingestellt *)
			END_IF;
			xStFct_StartMainPrc:=FALSE;
			xStFct_InitStep:=FALSE;
			iStFct_StepPrc:=iStFct_StepPrc + 1;
		END_IF;
	3:	IF NOT(xStFct_StartPrc_Parallel) THEN
			T_Station_Work.THWWorkStation.TCtrlWork.xZAxisBrakeBlocked:=xStFct_ZAxisBrakeBlocked;
			T_Station_Work.THWWorkStation.TCtrlWork.xBlockCheckAxisBrake:=FALSE;
			xStFct_StartMainPrc:=FALSE;
			xStFct_InitStep:=FALSE;
			iStFct_StepPrc:=0;
			xStFct_SetEnd:=TRUE;
		END_IF;
	END_CASE;
END_IF;
(******************************************************************************************************************************************)
(****************************			             Stationsfunktion Parallelablauf                                       *****************************)
(******************************************************************************************************************************************)
IF xStFct_StartPrc_Parallel AND NOT(xStFct_SetEnd) AND NOT(xStFct_HardwareError) THEN
	CASE iStFct_StepPrc_Parallel OF
	1:	iStFct_StepPrc_Parallel:=1;
		xStFct_InitStep_Parallel:=FALSE;
		xStFct_StartPrc_Parallel:=FALSE;
	END_CASE;
END_IF;
(******************************************************************************************************************************************)
(****************************				     Stationsfunktion Endprozedur                                    *****************************)
(******************************************************************************************************************************************)
StationFunction_Ctrl_End;
END_ACTION
ACTION StationFunction_Fct_11_Centring:
(******************************************************************************************************************************************)
(****************************				           Reset Stationsfunktion                                            *****************************)
(******************************************************************************************************************************************)
StationFunction_Ctrl_Reset;
(******************************************************************************************************************************************)
(****************************			        Stationsfunktion Fehler Controller                                    *****************************)
(******************************************************************************************************************************************)
StationFunction_Ctrl_Error;
(******************************************************************************************************************************************)
(****************************				    Stationsfunktion Haupt Controller                               *****************************)
(******************************************************************************************************************************************)
StationFunction_Ctrl_Main;
(******************************************************************************************************************************************)
(****************************			         Stationsfunktion sofort Unterbrechung                           *****************************)
(******************************************************************************************************************************************)
StationFunction_Ctrl_Stop;
(******************************************************************************************************************************************)
(****************************			             Stationsfunktion Hauptablauf                                       *****************************)
(******************************************************************************************************************************************)
IF xStFct_StartMainPrc AND NOT(xStFct_SetEnd) AND NOT(xStFct_HardwareError) AND NOT(xStFct_TmpStop) THEN
(***************************************************************************************************************************************************)
(* Überwachung auf die Axiale Auslenkung *)
	IF xStFct_ToolDeflectionActiv THEN
		IF NOT(IxToolDeflection2_St1) THEN
			xStFct_ToolDeflectionActiv:=FALSE;
			xStFct_InitAxialSensor:=FALSE;
			xStFct_CheckAxialSensor:=FALSE;
		END_IF;
	END_IF;
	IF (IxToolDeflection2_St1 OR xStFct_CheckAxialSensor) AND NOT(xStFct_ToolDeflectionActiv) THEN
		IF NOT(xStFct_InitAxialSensor) THEN
			xStFct_InitAxialSensor:=TRUE;
			xStFct_CheckAxialSensor:=TRUE;
			lrStFct_ActualPosition:=ptrTAxisZ^.T_LiveValue.lrActualPosition;
		END_IF;
		IF NOT(IxToolDeflection2_St1) THEN
			xStFct_InitAxialSensor:=FALSE;
			xStFct_CheckAxialSensor:=FALSE;
			xStFct_ToolDeflectionActiv:=FALSE;
		END_IF;
		IF (ABS(ptrTAxisZ^.T_LiveValue.lrActualPosition - lrStFct_ActualPosition) >= T_Station_Parameter.T_StProcess.rCenteringDeflectionSensorOffset) AND IxToolDeflection2_St1 THEN
			xStFct_ToolDeflectionActiv:=TRUE;
		END_IF;
	END_IF;
(***************************************************************************************************************************************************)
(* Hauptablauf für das Zentrieren *)
	CASE iStFct_StepPrc OF
	(* ZylAuslenkung mit ZentrierKraft setzen *)
	(* ZylWPUnfix setzen *)
	1:	gxWP_Analyse_ActiveCentering:=TRUE;
		lrZ1HCMinPosition:=0.0;
		lrZ1HCMaxPosition:=0.0;
		diHCCheckCounter:=0;
		T_ExchgParam.T_StationCommon.diCentringNumberHCinWindow:=0;
		wStFct_Status:=0;
		xZFastSpeedSettled:=FALSE;
		IF gxHardwareOFF OR gxAxisOFF THEN
			gxWP_Analyse_ActiveWork:=TRUE;
			xStFct_StartMainPrc:=FALSE;
			xStFct_InitStep:=FALSE;
			iStFct_StepPrc:=90;
			IF NOT(IxCylWPUnfixAtWorkPos_St1) THEN
				xStFct_HardwareError:=TRUE;
				diStFct_TmpErrorNr:=30;	(* Beim Zentrieren muss der ZylWstkEntspannen auf BearbeitPos sein *)
				RETURN;
			END_IF;
			RETURN;
		END_IF;
		(* Überprüfmechanismen die bestehen müssen, damit diese Funktion gestartet werden kann *)
		IF NOT(ptrTAxisZ^.T_CtrleSingle.xRef) THEN	(* Z Achse muss referenziert sein *)
			xStFct_HardwareError:=TRUE;
			diStFct_TmpErrorNr:=9;	(* Z Achse muss referenziert sein *)
			RETURN;
		END_IF;
		(* Überprüfe alle Positionen der Z Achse *)
		StationFunction_Ctrl_CheckPos_Z;
		IF xStFct_PositionOutRange_Z THEN
			xStFct_HardwareError:=TRUE;
			diStFct_TmpErrorNr:=iStFct_PosErrorNr;
			RETURN;
		END_IF;
		IF (garPositionEndProcCalc[1] > T_Station_Parameter.T_StProcess.rPositionEndMech) THEN
			xStFct_HardwareError:=TRUE;
			diStFct_TmpErrorNr:=12;		(* Hubprozesslänge > Z Mech EndPos *)
			RETURN;
		END_IF;
		IF (garCentringEndProcCalc[1] > T_Station_Parameter.T_StProcess.rPositionEndMech) THEN
			xStFct_HardwareError:=TRUE;
			diStFct_TmpErrorNr:=18;		(* Zentrier EndPos > Z Mech EndPos *)
			RETURN;
		END_IF;
		IF (garCentringEndProcCalc[1] > T_Station_Parameter.T_StProcess.rPositionEndProcMaxInc) AND T_Station_Parameter.T_StProcess.xCentringEndProcIncOnOff THEN
			xStFct_HardwareError:=TRUE;
			diStFct_TmpErrorNr:=19;			(* Z ZentrierPos berechn. > Z Bearb EndPos Max *)
			RETURN;
		END_IF;
		(* Überprüfe ob Wz im Wstk eingefädelt ist *)
		IF NOT(ptrTAxisZ^.T_LiveValue.lrActualPosition >= (grZ_WorkStartPos - 0.1)) THEN
			xStFct_HardwareError:=TRUE;
			diStFct_TmpErrorNr:=14;		(* Werkzeug ist nicht im Werkstück eingefädelt *)
			RETURN;
		END_IF;
		(* Überprüfmechanismen die bestehen müssen, damit diese Funktion gestartet werden kann *)
		IF NOT(IxCylWPUnfixAtWorkPos_St1) THEN
			xStFct_HardwareError:=TRUE;
			diStFct_TmpErrorNr:=30;	(* Beim Zentrieren muss der ZylWstkEntspannen auf BearbeitPos sein *)
			RETURN;
		END_IF;
		IF NOT(xStFct_InitStep) THEN
			xStFct_InitStep:=TRUE;
			IF NOT(ptrTAxisS^.T_CtrleSingle.xPower) THEN
				ptrTAxisS^.T_CtrleSingle.iFunction:=3;	(* Strom einschalten *)
				ptrTAxisS^.T_CtrleSingle.xExecute:=TRUE;
			END_IF;
			(* Zylinder für Auslenkung-->mit Zentrierkraft *)
			ptrTCylToolDeflection^.T_CtrleCyl.iFunction:=2;
			ptrTCylToolDeflection^.T_Config.tDelayOn:=T#0.3s;
			ptrTCylToolDeflection^.T_CtrleCyl.T_Analog.rForceIn:=T_Station_Parameter.T_StProcess.rCentringForceDeflection;
			ptrTCylToolDeflection^.T_CtrleCyl.xExecute:=TRUE;
			QxCylWPUnfix_St1:=TRUE;		(* Wstk Spannung lösen *)
		END_IF;
		IF NOT(ptrTCylToolDeflection^.T_CtrleCyl.xExecute) AND ptrTCylToolDeflection^.T_CtrleCyl.xDone THEN
			xStFct_StartMainPrc:=FALSE;
			xStFct_InitStep:=FALSE;
			iStFct_StepPrc:=iStFct_StepPrc + 1;
		END_IF
	(* Z1 Achse auf ZentrierPos fahren -->Zentriergeschwindigkeit setzen *)
	(* S Achse mit ZentrierGeschwindigkeit *)
	(* O Achse mit ZentrierGeschwindigkeit *)
	2:	IF NOT(xStFct_InitStep) THEN
			xStFct_InitStep:=TRUE;
			ptrTAxisZ^.T_CtrleSingle.iFunction:=7;	(* Absolut Bewegung *)
			ptrTAxisZ^.T_CtrleSingle.lrPosition:=garCentringEndProcCalc[1];				(* Z1 Achse auf ZentrierPos fahren *)
			ptrTAxisZ^.T_CtrleSingle.lrVelocity:=T_Station_Parameter.T_StProcess.rCentringPosSpeedFastZ1Axis;	(* Mit schneller Zentriergeschwindigkeit fahren *)
			ptrTAxisZ^.T_CtrleSingle.xExecute:=TRUE;
			IF (T_Station_Parameter.T_StProcess.rCentringSpeedSAxis <> 0.0) THEN
				(* Spindel mit Einfädelgeschwindigkeit *)
				IF ptrTAxisS^.T_CtrleSingle.xNotMoving THEN
					ptrTAxisS^.T_CtrleSingle.iFunction:=6;	(* Move Velocity *)
				ELSE
					ptrTAxisS^.T_CtrleSingle.iFunction:=12;	(* Move Velocity *)
				END_IF;
				ptrTAxisS^.T_CtrleSingle.lrVelocity:=T_Station_Parameter.T_StProcess.rCentringSpeedSAxis;
				ptrTAxisS^.T_CtrleSingle.xExecute:=TRUE;
			ELSE
				IF (NOT(ptrTAxisS^.T_CtrleSingle.xNotMoving) OR NOT(ptrTAxisS^.T_CtrleSingle.xDone))
				AND NOT((ptrTAxisS^.T_CtrleSingle.iFunction = 5) AND NOT(ptrTAxisS^.T_CtrleSingle.xDone)) AND NOT(ptrTAxisS^.T_CtrleSingle.xErr) THEN
					ptrTAxisS^.T_CtrleSingle.iFunction:=5;
					ptrTAxisS^.T_CtrleSingle.xExecute:=TRUE;
				END_IF;
			END_IF
			IF (T_Station_Parameter.T_StProcess.rCentringSpeedOAxis > 0.0) THEN
				QxFastStrokeOn_St1:=TRUE;
				QiAFastStroke:=REAL_TO_INT(32757 / 50.0 * T_Station_Parameter.T_StProcess.rCentringSpeedOAxis);		(* 32767digits / 50Hz * Param Hz *)
			END_IF;
		END_IF;
		IF TRUE THEN
			xStFct_StartMainPrc:=FALSE;
			xStFct_InitStep:=FALSE;
			iStFct_StepPrc:=iStFct_StepPrc + 1;
		END_IF;
	(* Der erste HC im Schnellgang wird gesucht *)
	3:	IF ptrTCylToolDeflection^.T_CtrleCyl.xStatePosOn AND NOT(xStFct_StopSlide) THEN	(* Neu wird der HC1 auch überwacht und falls eintrifft dann stoppen und z auf LadePos setzen und Fehler ausgeben *)
			xStFct_StopSlide:=TRUE;
			wStFct_Status:=1;	(* 1 = < Wz Auslenk. Sensor > *)
			lrActualPositionSaveSwitchZSpeed:=ptrTAxisZ^.T_LiveValue.lrActualPosition;
		END_IF;
		IF xStFct_ToolDeflectionActiv AND NOT(xStFct_StopSlide) THEN
			xStFct_StopSlide:=TRUE;
			wStFct_Status:=5;	(* 1 = < Wz Auslenk 2. Sensor > *)
			lrActualPositionSaveSwitchZSpeed:=ptrTAxisZ^.T_LiveValue.lrActualPosition;
		END_IF;
		IF NOT(ptrTAxisZ^.T_CtrleSingle.xExecute) AND ptrTAxisZ^.T_CtrleSingle.xDone THEN
			(* Wz konnte erfolgreich Zentriert werden aber es hatte keinen HC *)
			iStFct_StepPrc:=50;		(* Z Achse um einen Offset zurückfahren oder auf LadePosition zurücksetzen *)
			xStFct_StartMainPrc:=FALSE;
			xStFct_InitStep:=FALSE;
			IF T_Station_Parameter.T_StProcess.xCentringEndProcIncOnOff THEN
				garCentringEndProcCalc[1]:=garCentringEndProcCalc[1] + T_Station_Parameter.T_StProcess.rCentringEndProInc;	(* Zentrier EndPos Inkrementieren *)
			END_IF;
			RETURN;
		END_IF;
		IF xStFct_StopSlide AND NOT(ptrTAxisZ^.T_CtrleSingle.xExecute) AND NOT(ptrTAxisZ^.T_CtrleSingle.xDone) AND
		    NOT(ptrTAxisZ^.T_CtrleSingle.xNotMoving) AND (ptrTAxisZ^.T_CtrleSingle.iFunction <> 12) THEN
			ptrTAxisZ^.T_CtrleSingle.iFunction:=5;
			ptrTAxisZ^.T_CtrleSingle.xExecute:=TRUE;
			(* init. variable *)
			xStFct_StopSlide:=FALSE;
			iStFct_StepPrc:=iStFct_StepPrc + 1;
			xStFct_InitStep:=FALSE;
		END_IF;
	4:	(* Abwarten bis die HubAchse stillsteht *)
		IF NOT(ptrTAxisZ^.T_CtrleSingle.xExecute) AND ptrTAxisZ^.T_CtrleSingle.xDone THEN
			xStFct_StartMainPrc:=FALSE;
			xStFct_InitStep:=FALSE;
			IF (wStFct_Status <> 1) THEN
				iStFct_StepPrc:=iStFct_StepPrc + 1;
			ELSE
				iStFct_StepPrc:=50;	(* Wenn HC1 eintrifft dann auf LadePos zurück und Fehler ausgeben *)
			END_IF;
		END_IF;
	5:	(* Z Achse um einen Offset beim ersten HC zurücksetzen *)
		IF NOT(xStFct_InitStep) THEN
			xStFct_InitStep:=TRUE;
			IF ((ptrTAxisZ^.T_LiveValue.lrActualPosition - ABS(T_Station_Parameter.T_StProcess.rCentringBackStrokeOffsetFirstHC)) >= grZ_WorkStartPos) THEN
				ptrTAxisZ^.T_CtrleSingle.iFunction:=8;
				ptrTAxisZ^.T_CtrleSingle.lrDistance:=T_Station_Parameter.T_StProcess.rCentringBackStrokeOffsetFirstHC;
				ptrTAxisZ^.T_CtrleSingle.lrVelocity:=T_Station_Parameter.T_StProcess.rCentringBackStrokeSpeed;
			ELSE
				ptrTAxisZ^.T_CtrleSingle.iFunction:=7;
				ptrTAxisZ^.T_CtrleSingle.lrPosition:=grZ_WorkStartPos;
				ptrTAxisZ^.T_CtrleSingle.lrVelocity:=T_Station_Parameter.T_StProcess.rCentringBackStrokeSpeed;
			END_IF;
			ptrTAxisZ^.T_CtrleSingle.xExecute:=TRUE;
		END_IF;
		IF NOT(ptrTAxisZ^.T_CtrleSingle.xExecute) AND ptrTAxisZ^.T_CtrleSingle.xDone THEN
			xStFct_StartMainPrc:=FALSE;
			xStFct_InitStep:=FALSE;
			iStFct_StepPrc:=iStFct_StepPrc + 5;
		END_IF;

	10:	(* Z Achse auf Zentrierposition mit langsamer Geschwindigkeit setzen *)
		IF NOT(xStFct_InitStep) THEN
			xStFct_InitStep:=TRUE;
			ptrTAxisZ^.T_CtrleSingle.iFunction:=7;	(* Absolut Bewegung *)
			ptrTAxisZ^.T_CtrleSingle.lrPosition:=garCentringEndProcCalc[1];				(* Z1 Achse auf ZentrierPos fahren *)
			ptrTAxisZ^.T_CtrleSingle.lrVelocity:=T_Station_Parameter.T_StProcess.rCentringPosSpeedSlowZ1Axis;	(* Mit langsamer Zentriergeschwindigkeit fahren *)
			ptrTAxisZ^.T_CtrleSingle.xExecute:=TRUE;
		END_IF;
		IF TRUE THEN
			xStFct_StartMainPrc:=FALSE;
			xStFct_InitStep:=FALSE;
			iStFct_StepPrc:=iStFct_StepPrc + 1;
		END_IF;
	(* Die weiteren HC im Langsamgang wird gesucht *)
	11:	IF ptrTCylToolDeflection^.T_CtrleCyl.xStatePosOn AND NOT(xStFct_StopSlide) THEN	(* Neu wird der HC1 auch überwacht und falls eintrifft dann stoppen und z auf LadePos setzen und Fehler ausgeben *)
			xStFct_StopSlide:=TRUE;
			wStFct_Status:=1;	(* 1 = < Wz Auslenk. Sensor > *)
			T_Station_Work.THWWorkStation.TCtrlWork.iOverLimitCounterCentering:=T_Station_Work.THWWorkStation.TCtrlWork.iOverLimitCounterCentering + 1;	(* Erst hier werden die HC gezählt, d.h. der erste wird nicht gezählt *)
			lrActualPositionSave:=ptrTAxisZ^.T_LiveValue.lrActualPosition;
			lrActualPositionSaveSwitchZSpeed:=ptrTAxisZ^.T_LiveValue.lrActualPosition;
			xZFastSpeedSettled:=FALSE;
		END_IF;
		IF xStFct_ToolDeflectionActiv AND NOT(xStFct_StopSlide) THEN
			xStFct_StopSlide:=TRUE;
			wStFct_Status:=5;	(* 1 = < Wz Auslenk 2. Sensor > *)
			T_Station_Work.THWWorkStation.TCtrlWork.iOverLimitCounterCentering:=T_Station_Work.THWWorkStation.TCtrlWork.iOverLimitCounterCentering + 1;	(* Erst hier werden die HC gezählt, d.h. der erste wird nicht gezählt *)
			lrActualPositionSave:=ptrTAxisZ^.T_LiveValue.lrActualPosition;
			lrActualPositionSaveSwitchZSpeed:=ptrTAxisZ^.T_LiveValue.lrActualPosition;
			xZFastSpeedSettled:=FALSE;
		END_IF;
		IF NOT(ptrTAxisZ^.T_CtrleSingle.xExecute) AND ptrTAxisZ^.T_CtrleSingle.xDone THEN
			(* Wz konnte erfolgreich Zentriert werden und es hatte mindesten einen HC *)
			xZFastSpeedSettled:=FALSE;
			wStFct_Status:=0;
			iStFct_StepPrc:=50;		(* Z Achse um einen Offset zurückfahren oder auf LadePosition zurücksetzen *)
			xStFct_StartMainPrc:=FALSE;
			xStFct_InitStep:=FALSE;
			IF T_Station_Parameter.T_StProcess.xCentringEndProcIncOnOff THEN
				garCentringEndProcCalc[1]:=garCentringEndProcCalc[1] + T_Station_Parameter.T_StProcess.rCentringEndProInc;	(* Zentrier EndPos Inkrementieren *)
			END_IF;
			RETURN;
		END_IF;
		IF xStFct_StopSlide AND NOT(ptrTAxisZ^.T_CtrleSingle.xExecute) AND NOT(ptrTAxisZ^.T_CtrleSingle.xDone) AND
		    NOT(ptrTAxisZ^.T_CtrleSingle.xNotMoving) AND (ptrTAxisZ^.T_CtrleSingle.iFunction <> 12) THEN
			ptrTAxisZ^.T_CtrleSingle.iFunction:=5;
			ptrTAxisZ^.T_CtrleSingle.xExecute:=TRUE;
			(* init. variable *)
			xStFct_StopSlide:=FALSE;
			iStFct_StepPrc:=iStFct_StepPrc + 1;
			xStFct_InitStep:=FALSE;
			xZFastSpeedSettled:=FALSE;
			RETURN;
		END_IF;
		IF NOT(xStFct_StopSlide) AND NOT(ptrTAxisZ^.T_CtrleSingle.xExecute) AND NOT(ptrTAxisZ^.T_CtrleSingle.xDone) AND
		    NOT(ptrTAxisZ^.T_CtrleSingle.xNotMoving) AND (ptrTAxisZ^.T_CtrleSingle.iFunction <> 12) AND NOT(xZFastSpeedSettled) THEN
			IF (ptrTAxisZ^.T_LiveValue.lrActualPosition >= (lrActualPositionSaveSwitchZSpeed + T_Station_Parameter.T_StProcess.rCentringOffsetSlowToFastZSpeed)) AND (T_Station_Parameter.T_StProcess.rCentringOffsetSlowToFastZSpeed <> 0.0) THEN
				(* Wenn die Z Achse um einen definierten Offset kein HC eingetroffen ist, dann soll es auf die schnelle Geschwindigkeit umschalten *)
				xZFastSpeedSettled:=TRUE;
				ptrTAxisZ^.T_CtrleSingle.iFunction:=12;	(* Move Velocity *)
				ptrTAxisZ^.T_CtrleSingle.lrVelocity:=T_Station_Parameter.T_StProcess.rCentringPosSpeedFastZ1Axis;
				ptrTAxisZ^.T_CtrleSingle.xExecute:=TRUE;
			END_IF;
		END_IF;
	12:	(* Abwarten bis die HubAchse stillsteht *)
		IF NOT(ptrTAxisZ^.T_CtrleSingle.xExecute) AND ptrTAxisZ^.T_CtrleSingle.xDone THEN
			xStFct_StartMainPrc:=FALSE;
			xStFct_InitStep:=FALSE;
			TONWaitHCActive(IN:=FALSE);
			TONWaitHCInactive(IN:=FALSE);
			IF (wStFct_Status <> 1) THEN
				IF (lrZ1HCMinPosition = 0) THEN
					lrZ1HCMinPosition:=lrActualPositionSave;
					lrZ1HCMaxPosition:=lrActualPositionSave;
					IF (T_Station_Parameter.T_StProcess.iCentringSelectProcess <= 1) THEN
						iStFct_StepPrc:=iStFct_StepPrc + 1;	(* Konventioneller Ablauf *)
					ELSE
						iStFct_StepPrc:=iStFct_StepPrc + 3;	(* Ablauf für Finde Grauzone, zurückfahren bis HC2 nicht mehr angibt *)
					END_IF;
				ELSE
					IF (lrActualPositionSave < lrZ1HCMinPosition) THEN
						lrZ1HCMinPosition:=lrActualPositionSave;
					END_IF;
					IF (lrActualPositionSave > lrZ1HCMaxPosition) THEN
						lrZ1HCMaxPosition:=lrActualPositionSave;
					END_IF;
					IF ((lrZ1HCMaxPosition - lrZ1HCMinPosition) <= T_Station_Parameter.T_StProcess.rCentringHCWindow) THEN
						diHCCheckCounter:=diHCCheckCounter + 1;
						IF (diHCCheckCounter >= T_Station_Parameter.T_StProcess.iCentringNumberMaxHCinWindow) THEN
							IF (T_Station_Parameter.T_StProcess.iCentringSelectProcess <= 1) THEN
								(* Maximale Anzahl HC im definierten Fenster erreicht und der Prozess wird abegbrochen *)
								wStFct_Status:=99;
								iStFct_StepPrc:=50;
							ELSE
								(* Neu definiert Prozessablauf für Finde Grauzone. hier wird nicht abgebrochen sondern Rückhub wie bei normalen Ablauf *)
								iStFct_StepPrc:=20;
							END_IF;
						ELSE
							IF (T_Station_Parameter.T_StProcess.iCentringSelectProcess <= 1) THEN
								iStFct_StepPrc:=iStFct_StepPrc + 1;	(* Konventioneller Ablauf *)
							ELSE
								iStFct_StepPrc:=iStFct_StepPrc + 3;	(* Ablauf für Finde Grauzone, zurückfahren bis HC2 nicht mehr angibt *)
							END_IF;
						END_IF;
					ELSE
						diHCCheckCounter:=0;
						lrZ1HCMinPosition:=lrActualPositionSave;
						lrZ1HCMaxPosition:=lrActualPositionSave;
						IF (T_Station_Parameter.T_StProcess.iCentringSelectProcess <= 1) THEN
							iStFct_StepPrc:=iStFct_StepPrc + 1;
						ELSE
							iStFct_StepPrc:=iStFct_StepPrc + 3;	(* Ablauf für Finde Grauzone, zurückfahren bis HC2 nicht mehr angibt *)
						END_IF;
					END_IF;
				END_IF;
			ELSE
				iStFct_StepPrc:=50;	(* Wenn HC1 eintrifft dann auf LadePos zurück und Fehler ausgeben *)
			END_IF;
		END_IF;
		T_ExchgParam.T_StationCommon.diCentringNumberHCinWindow:=diHCCheckCounter;
	13:	(* Wartezeiten laufen lassen *)
		TONWaitHCActive(IN:=TRUE,PT:=REAL_TO_TIME(T_Station_Parameter.T_StProcess.rCentringTimeHCActive * 1000.0));
		TONWaitHCInactive(IN:=NOT(IxToolDeflection2_St1),PT:=REAL_TO_TIME(T_Station_Parameter.T_StProcess.rCentringTimeHCInactive * 1000.0));
		IF TONWaitHCInactive.Q THEN
			(* HC ist für eine bestimmte Zeit nicht mehr Aktiv und deshalb kann die Z Achse wieder weiterfahren im Langsamgang *)
			xStFct_ToolDeflectionActiv:=FALSE;
			xStFct_StartMainPrc:=FALSE;
			xStFct_InitStep:=FALSE;
			iStFct_StepPrc:=iStFct_StepPrc - 3 ;
			RETURN;
		END_IF;
		IF TONWaitHCActive.Q THEN
			(* HC ist immer noch Aktiv, dann muss die Z Achse um einen Offset zurückgesetzt werden *)
			xStFct_StartMainPrc:=FALSE;
			xStFct_InitStep:=FALSE;
			iStFct_StepPrc:=iStFct_StepPrc + 7;
		END_IF;

	(* Gilt nur für den Zentrierablauf mit Finde Grauzone, nach dem ersten HC zurückfahren bis HC nicht mehr eintrifft und dann Normal wieder langsam nach vorne fahren *)
	15:	IF NOT(xStFct_InitStep) THEN
			xStFct_InitStep:=TRUE;
			ptrTAxisZ^.T_CtrleSingle.iFunction:=7;	(* Absolut Bewegung *)
			ptrTAxisZ^.T_CtrleSingle.lrPosition:=grZ_WorkStartPos;	(* Zurück bis Startpos fahren und soabld HC2 nicht mehr aktiv ist kann gestoppt werden *)
			ptrTAxisZ^.T_CtrleSingle.lrVelocity:=T_Station_Parameter.T_StProcess.rCentringPosSpeedSlowZ1Axis;	(* Mit langsamer Zentriergeschwindigkeit fahren *)
			ptrTAxisZ^.T_CtrleSingle.xExecute:=TRUE;
			TONWaitHCInactive(IN:=FALSE);
		END_IF;
		IF TRUE THEN
			xStFct_StartMainPrc:=FALSE;
			xStFct_InitStep:=FALSE;
			iStFct_StepPrc:=iStFct_StepPrc + 1;
		END_IF;
	16:	TONWaitHCInactive(IN:=NOT(IxToolDeflection2_St1),PT:=REAL_TO_TIME(T_Station_Parameter.T_StProcess.rCentringTimeHCInactive * 1000.0));
		IF TONWaitHCInactive.Q THEN
			(* HC ist für eine bestimmte Zeit nicht mehr Aktiv und deshalb kann die Z Achse wieder weiterfahren im Langsamgang *)
			xStFct_ToolDeflectionActiv:=FALSE;
			xStFct_StartMainPrc:=FALSE;
			xStFct_InitStep:=FALSE;
			xStFct_StopSlide:=TRUE;
		END_IF;
		IF xStFct_StopSlide AND NOT(ptrTAxisZ^.T_CtrleSingle.xExecute) AND NOT(ptrTAxisZ^.T_CtrleSingle.xDone) AND
		    NOT(ptrTAxisZ^.T_CtrleSingle.xNotMoving) AND (ptrTAxisZ^.T_CtrleSingle.iFunction <> 12) THEN
			ptrTAxisZ^.T_CtrleSingle.iFunction:=5;
			ptrTAxisZ^.T_CtrleSingle.xExecute:=TRUE;
			(* init. variable *)
			xStFct_StopSlide:=FALSE;
			iStFct_StepPrc:=iStFct_StepPrc + 1;
			xStFct_InitStep:=FALSE;
		END_IF;
		IF NOT(ptrTAxisZ^.T_CtrleSingle.xExecute) AND ptrTAxisZ^.T_CtrleSingle.xDone THEN
			(* Der HC2 ist immer noch aktiv und die Startposition wurde erreicht und es muss einen Fehler ausgegeben werden *)
			iStFct_StepPrc:=50;		(* Z Achse um einen Offset zurückfahren oder auf LadePosition zurücksetzen *)
			xStFct_StartMainPrc:=FALSE;
			xStFct_InitStep:=FALSE;
			wStFct_Status:=98;	(* Dummy Zahl setzen um es auffangen zu können *)
			RETURN;
		END_IF;
	17:	(* Abwarten bis die HubAchse stillsteht *)
		IF NOT(ptrTAxisZ^.T_CtrleSingle.xExecute) AND ptrTAxisZ^.T_CtrleSingle.xDone THEN
			xStFct_ToolDeflectionActiv:=FALSE;
			xStFct_StartMainPrc:=FALSE;
			xStFct_InitStep:=FALSE;
			iStFct_StepPrc:=iStFct_StepPrc - 7 ;
			RETURN;
		END_IF;

	20:	(* Z Achse um einen Offset nach dem ersten HC zurücksetzen *)
		IF NOT(xStFct_InitStep) THEN
			xStFct_InitStep:=TRUE;
			IF ((ptrTAxisZ^.T_LiveValue.lrActualPosition - ABS(T_Station_Parameter.T_StProcess.rCentringBackStrokeOffsetAfterFirstHC)) >= grZ_WorkStartPos) THEN
				ptrTAxisZ^.T_CtrleSingle.iFunction:=8;
				ptrTAxisZ^.T_CtrleSingle.lrDistance:=T_Station_Parameter.T_StProcess.rCentringBackStrokeOffsetAfterFirstHC;
				ptrTAxisZ^.T_CtrleSingle.lrVelocity:=T_Station_Parameter.T_StProcess.rCentringBackStrokeSpeed;
			ELSE
				ptrTAxisZ^.T_CtrleSingle.iFunction:=7;
				ptrTAxisZ^.T_CtrleSingle.lrPosition:=grZ_WorkStartPos;
				ptrTAxisZ^.T_CtrleSingle.lrVelocity:=T_Station_Parameter.T_StProcess.rCentringBackStrokeSpeed;
			END_IF;
			ptrTAxisZ^.T_CtrleSingle.xExecute:=TRUE;
		END_IF;
		IF NOT(ptrTAxisZ^.T_CtrleSingle.xExecute) AND ptrTAxisZ^.T_CtrleSingle.xDone THEN
			xStFct_StartMainPrc:=FALSE;
			xStFct_InitStep:=FALSE;
			iStFct_StepPrc:=iStFct_StepPrc + 1;
		END_IF;
	21:	(* Z Achse im Schnellgang zum letzte HC minus den Offset setzen *)
		IF NOT(xStFct_InitStep) THEN
			xStFct_InitStep:=TRUE;
			ptrTAxisZ^.T_CtrleSingle.iFunction:=7;	(* Absolut Bewegung *)
			ptrTAxisZ^.T_CtrleSingle.lrPosition:=lrActualPositionSave - ABS(T_Station_Parameter.T_StProcess.rCentringOffsetBeforeLastHC);	(* Z1 Achse auf die letzte HC Position minus den Offset setzen *)
			ptrTAxisZ^.T_CtrleSingle.lrVelocity:=T_Station_Parameter.T_StProcess.rCentringPosSpeedFastZ1Axis;							(* Mit schneller Zentriergeschwindigkeit fahren *)
			ptrTAxisZ^.T_CtrleSingle.xExecute:=TRUE;
		END_IF;
		IF ptrTCylToolDeflection^.T_CtrleCyl.xStatePosOn AND NOT(xStFct_StopSlide) THEN	(* Neu wird der HC1 auch überwacht und falls eintrifft dann stoppen und z auf LadePos setzen und Fehler ausgeben *)
			xStFct_StopSlide:=TRUE;
			wStFct_Status:=1;	(* 1 = < Wz Auslenk. Sensor > *)
		END_IF;
		IF xStFct_ToolDeflectionActiv AND NOT(xStFct_StopSlide) THEN	(* Trotzdem überwachen ob die Auslenkung angeben sollte *)
			xStFct_StopSlide:=TRUE;
		END_IF;
		IF NOT(ptrTAxisZ^.T_CtrleSingle.xExecute) AND ptrTAxisZ^.T_CtrleSingle.xDone THEN
			(* Die Z Achse kann wieder weiterfahren im Langsamgang *)
			xStFct_StartMainPrc:=FALSE;
			xStFct_InitStep:=FALSE;
			iStFct_StepPrc:=iStFct_StepPrc - 11 ;
		END_IF;
		IF xStFct_StopSlide AND NOT(ptrTAxisZ^.T_CtrleSingle.xExecute) AND NOT(ptrTAxisZ^.T_CtrleSingle.xDone) AND
		    NOT(ptrTAxisZ^.T_CtrleSingle.xNotMoving) AND (ptrTAxisZ^.T_CtrleSingle.iFunction <> 12) THEN
			ptrTAxisZ^.T_CtrleSingle.iFunction:=5;
			ptrTAxisZ^.T_CtrleSingle.xExecute:=TRUE;
			(* init. variable *)
			xStFct_StopSlide:=FALSE;
			iStFct_StepPrc:=iStFct_StepPrc + 1;
			xStFct_InitStep:=FALSE;
		END_IF;
	22:	(* Abwarten bis die HubAchse stillsteht *)
		IF NOT(ptrTAxisZ^.T_CtrleSingle.xExecute) AND ptrTAxisZ^.T_CtrleSingle.xDone THEN
			xStFct_StartMainPrc:=FALSE;
			xStFct_InitStep:=FALSE;
			IF (wStFct_Status <> 1) THEN
				iStFct_StepPrc:=iStFct_StepPrc - 17;
			ELSE
				iStFct_StepPrc:=50;	(* Wenn HC1 eintrifft dann auf LadePos zurück und Fehler ausgeben *)
			END_IF;
		END_IF;

